C03633=1059.464,137.900,419.147,172.001,31.225,155.799
C03634=1059.459,137.652,419.168,172.000,31.222,155.799
C03635=1059.452,137.402,419.188,171.998,31.219,155.798
C03636=1059.447,137.154,419.210,171.997,31.217,155.798
C03637=1059.441,136.904,419.231,171.995,31.214,155.797
C03638=1059.435,136.656,419.251,171.993,31.211,155.797
C03639=1059.429,136.406,419.272,171.991,31.209,155.797
C03640=1059.423,136.157,419.293,171.989,31.206,155.796
C03641=1059.417,135.909,419.313,171.987,31.203,155.796
C03642=1059.411,135.659,419.334,171.986,31.201,155.795
C03643=1059.405,135.411,419.355,171.984,31.198,155.795
C03644=1059.399,135.161,419.376,171.983,31.196,155.794
C03645=1059.394,134.912,419.397,171.981,31.193,155.794
C03646=1059.387,134.663,419.417,171.979,31.190,155.794
C03647=1059.382,134.414,419.438,171.977,31.188,155.793
C03648=1059.376,134.165,419.459,171.976,31.185,155.793
C03649=1059.370,133.916,419.480,171.974,31.182,155.792
C03650=1059.364,133.666,419.500,171.972,31.180,155.792
C03651=1059.357,133.418,419.521,171.970,31.177,155.792
C03652=1059.352,133.168,419.542,171.968,31.174,155.791
C03653=1059.347,132.919,419.562,171.967,31.172,155.791
C03654=1059.340,132.670,419.583,171.966,31.169,155.790
C03655=1059.335,132.421,419.604,171.964,31.167,155.790
C03656=1059.330,132.172,419.624,171.962,31.164,155.789
C03657=1059.323,131.923,419.645,171.960,31.161,155.789
C03658=1059.317,131.674,419.666,171.958,31.159,155.789
C03659=1059.311,131.425,419.686,171.956,31.157,155.788
C03660=1059.305,131.176,419.706,171.955,31.154,155.788
C03661=1059.299,130.927,419.728,171.954,31.151,155.787
C03662=1059.293,130.678,419.748,171.952,31.149,155.787
C03663=1059.287,130.429,419.768,171.950,31.146,155.787
C03664=1059.281,130.179,419.789,171.948,31.143,155.786
C03665=1059.275,129.930,419.809,171.946,31.141,155.786
C03666=1059.270,129.681,419.829,171.945,31.139,155.785
C03667=1059.263,129.432,419.850,171.943,31.136,155.785
C03668=1059.257,129.184,419.870,171.941,31.133,155.785
C03669=1059.251,128.934,419.891,171.939,31.131,155.784
C03670=1059.245,128.685,419.911,171.938,31.128,155.784
C03671=1059.239,128.436,419.931,171.936,31.126,155.783
C03672=1059.233,128.186,419.952,171.935,31.123,155.783
C03673=1059.227,127.937,419.972,171.933,31.120,155.783
C03674=1059.221,127.689,419.993,171.931,31.118,155.782
C03675=1059.215,127.439,420.014,171.929,31.116,155.782
C03676=1059.209,127.191,420.034,171.927,31.113,155.781
C03677=1059.203,126.942,420.054,171.926,31.110,155.781
C03678=1059.197,126.716,420.072,171.925,31.108,155.781
C03679=1059.192,126.489,420.091,171.923,31.106,155.780
C03680=1059.187,126.265,420.109,171.921,31.103,155.780
C03681=1059.181,126.039,420.128,171.920,31.101,155.780
C03682=1059.175,125.813,420.146,171.918,31.098,155.779
C03683=1059.170,125.587,420.164,171.916,31.096,155.779
C03684=1059.164,125.361,420.182,171.915,31.094,155.778
C03685=1059.160,125.136,420.200,171.914,31.092,155.778
C03686=1059.153,124.887,420.221,171.912,31.089,155.778
C03687=1059.147,124.638,420.241,171.910,31.086,155.777
C03688=1059.142,124.389,420.262,171.909,31.084,155.777
C03689=1059.136,124.139,420.282,171.907,31.081,155.776
C03690=1059.130,123.890,420.302,171.905,31.079,155.776
C03691=1059.124,123.641,420.322,171.904,31.076,155.776
C03692=1059.118,123.392,420.342,171.902,31.073,155.775
C03693=1059.112,123.143,420.362,171.900,31.071,155.775
C03694=1059.106,122.894,420.382,171.898,31.069,155.774
C03695=1059.100,122.645,420.403,171.897,31.066,155.774
C03696=1059.094,122.396,420.423,171.895,31.063,155.774
C03697=1059.088,122.146,420.443,171.894,31.061,155.773
C03698=1059.082,121.897,420.463,171.892,31.058,155.773
C03699=1059.077,121.648,420.484,171.890,31.055,155.772
C03700=1059.071,121.399,420.504,171.888,31.053,155.772
C03701=1059.065,121.151,420.524,171.887,31.050,155.772
C03702=1059.058,120.901,420.544,171.886,31.048,155.771
C03703=1059.053,120.651,420.564,171.884,31.045,155.771
C03704=1059.047,120.403,420.584,171.882,31.042,155.770
C03705=1059.041,120.154,420.604,171.880,31.040,155.770
C03706=1059.033,119.822,420.631,171.878,31.036,155.769
C03707=1059.026,119.491,420.657,171.876,31.033,155.769
C03708=1059.018,119.158,420.684,171.874,31.030,155.768
C03709=1059.010,118.828,420.711,171.872,31.026,155.768
C03710=1059.004,118.578,420.731,171.870,31.024,155.767
C03711=1058.999,118.329,420.750,171.868,31.021,155.767
C03712=1058.992,118.080,420.771,171.867,31.018,155.767
C03713=1058.986,117.831,420.791,171.865,31.016,155.766
C03714=1058.981,117.582,420.811,171.864,31.013,155.766
C03715=1058.975,117.333,420.831,171.862,31.011,155.765
C03716=1058.969,117.083,420.850,171.860,31.008,155.765
C03717=1058.963,116.835,420.870,171.858,31.005,155.764
C03718=1058.957,116.586,420.890,171.857,31.003,155.764
C03719=1058.951,116.336,420.911,171.855,31.000,155.764
C03720=1058.946,116.086,420.931,171.854,30.997,155.763
C03721=1058.940,115.838,420.950,171.852,30.995,155.763
C03722=1058.934,115.589,420.970,171.850,30.992,155.762
C03723=1058.928,115.339,420.990,171.849,30.989,155.762
C03724=1058.923,115.090,421.010,171.847,30.987,155.762
C03725=1058.917,114.841,421.030,171.846,30.984,155.761
C03726=1058.911,114.592,421.049,171.844,30.981,155.761
C03727=1058.905,114.343,421.069,171.842,30.979,155.760
C03728=1058.900,114.094,421.090,171.840,30.976,155.760
C03729=1058.893,113.844,421.110,171.839,30.973,155.759
C03730=1058.887,113.595,421.130,171.838,30.971,155.759
C03731=1058.882,113.346,421.149,171.836,30.969,155.759
C03732=1058.875,113.097,421.168,171.834,30.966,155.758
C03733=1058.869,112.848,421.188,171.832,30.964,155.758
C03734=1058.863,112.599,421.207,171.830,30.961,155.758
C03735=1058.857,112.350,421.227,171.830,30.958,155.757
C03736=1058.852,112.101,421.247,171.828,30.956,155.757
C03737=1058.845,111.851,421.267,171.826,30.953,155.756
C03738=1058.839,111.602,421.286,171.824,30.950,155.756
C03739=1058.833,111.353,421.306,171.822,30.948,155.756
C03740=1058.828,111.104,421.325,171.822,30.946,155.755
C03741=1058.822,110.855,421.345,171.820,30.943,155.755
C03742=1058.815,110.570,421.367,171.818,30.940,155.754
C03743=1058.808,110.285,421.390,171.816,30.937,155.754
C03744=1058.801,110.000,421.412,171.814,30.934,155.753
C03745=1058.794,109.716,421.435,171.813,30.932,155.753
C03746=1058.788,109.467,421.454,171.811,30.929,155.753
C03747=1058.782,109.217,421.473,171.809,30.926,155.752
C03748=1058.776,108.968,421.493,171.807,30.924,155.752
C03749=1058.771,108.719,421.512,171.805,30.921,155.751
C03750=1058.764,108.469,421.533,171.804,30.919,155.751
C03751=1058.758,108.220,421.551,171.803,30.916,155.751
C03752=1058.752,107.971,421.571,171.801,30.914,155.750
C03753=1058.746,107.722,421.590,171.799,30.911,155.750
C03754=1058.740,107.473,421.610,171.797,30.908,155.749
C03755=1058.734,107.224,421.630,171.796,30.906,155.749
C03756=1058.729,106.974,421.649,171.795,30.904,155.749
C03757=1058.722,106.725,421.668,171.793,30.901,155.748
C03758=1058.716,106.476,421.688,171.791,30.898,155.748
C03759=1058.710,106.227,421.707,171.790,30.896,155.747
C03760=1058.705,105.978,421.726,171.788,30.893,155.747
C03761=1058.699,105.729,421.746,171.786,30.891,155.747
C03762=1058.692,105.480,421.765,171.785,30.888,155.746
C03763=1058.687,105.230,421.784,171.783,30.886,155.746
C03764=1058.681,104.981,421.804,171.782,30.883,155.745
C03765=1058.675,104.732,421.823,171.780,30.881,155.745
C03766=1058.669,104.483,421.842,171.778,30.878,155.745
C03767=1058.663,104.234,421.862,171.777,30.875,155.744
C03768=1058.657,103.985,421.881,171.776,30.873,155.744
C03769=1058.651,103.735,421.900,171.774,30.871,155.743
C03770=1058.645,103.486,421.919,171.772,30.868,155.743
C03771=1058.639,103.237,421.939,171.770,30.865,155.743
C03772=1058.633,102.988,421.958,171.769,30.863,155.742
C03773=1058.627,102.738,421.977,171.768,30.860,155.742
C03774=1058.622,102.489,421.996,171.766,30.857,155.741
C03775=1058.615,102.240,422.016,171.764,30.855,155.741
C03776=1058.609,101.991,422.035,171.762,30.853,155.741
C03777=1058.604,101.742,422.054,171.761,30.850,155.740
C03778=1058.598,101.492,422.074,171.760,30.847,155.740
C03779=1058.591,101.243,422.092,171.758,30.845,155.739
C03780=1058.585,100.994,422.112,171.756,30.842,155.739
C03781=1058.580,100.745,422.131,171.755,30.840,155.739
C03782=1058.573,100.496,422.150,171.753,30.837,155.738
C03783=1058.568,100.247,422.169,171.752,30.835,155.738
C03784=1058.563,99.997,422.188,171.750,30.832,155.737
C03785=1058.556,99.748,422.207,171.748,30.829,155.737
C03786=1058.550,99.499,422.226,171.747,30.827,155.737
C03787=1058.544,99.250,422.245,171.745,30.825,155.736
C03788=1058.538,99.001,422.265,171.743,30.822,155.736
C03789=1058.532,98.752,422.283,171.742,30.819,155.736
C03790=1058.526,98.502,422.303,171.741,30.817,155.735
C03791=1058.520,98.253,422.321,171.739,30.815,155.735
C03792=1058.514,98.004,422.340,171.737,30.812,155.734
C03793=1058.507,97.755,422.359,171.735,30.809,155.734
C03794=1058.502,97.505,422.378,171.735,30.807,155.734
C03795=1058.495,97.256,422.397,171.733,30.805,155.733
C03796=1058.490,97.007,422.416,171.731,30.802,155.733
C03797=1058.483,96.758,422.435,171.729,30.799,155.732
C03798=1058.477,96.508,422.454,171.728,30.797,155.732
C03799=1058.471,96.259,422.473,171.727,30.794,155.732
C03800=1058.466,96.010,422.492,171.725,30.792,155.731
C03801=1058.460,95.761,422.510,171.723,30.789,155.731
C03802=1058.454,95.512,422.530,171.721,30.787,155.730
C03803=1058.447,95.263,422.548,171.720,30.784,155.730
C03804=1058.442,95.013,422.567,171.719,30.781,155.730
C03805=1058.435,94.764,422.586,171.717,30.779,155.729
C03806=1058.428,94.479,422.608,171.715,30.776,155.729
C03807=1058.422,94.195,422.630,171.713,30.773,155.728
C03808=1058.415,93.910,422.650,171.711,30.771,155.728
C03809=1058.408,93.625,422.672,171.710,30.767,155.727
C03810=1058.403,93.376,422.691,171.708,30.765,155.727
C03811=1058.397,93.127,422.710,171.707,30.763,155.727
C03812=1058.391,92.877,422.729,171.705,30.760,155.726
C03813=1058.384,92.628,422.748,171.703,30.757,155.726
C03814=1058.379,92.379,422.767,171.702,30.755,155.726
C03815=1058.372,92.130,422.786,171.701,30.752,155.725
C03816=1058.367,91.881,422.803,171.699,30.750,155.725
C03817=1058.361,91.631,422.822,171.697,30.747,155.724
C03818=1058.355,91.382,422.841,171.696,30.745,155.724
C03819=1058.349,91.133,422.860,171.695,30.742,155.724
C03820=1058.343,90.883,422.879,171.693,30.740,155.723
C03821=1058.338,90.635,422.898,171.691,30.737,155.723
C03822=1058.331,90.385,422.916,171.690,30.735,155.722
C03823=1058.325,90.136,422.934,171.688,30.732,155.722
C03824=1058.319,89.886,422.954,171.686,30.730,155.722
C03825=1058.313,89.637,422.972,171.685,30.727,155.721
C03826=1058.307,89.388,422.990,171.684,30.725,155.721
C03827=1058.300,89.138,423.009,171.682,30.722,155.720
C03828=1058.295,88.890,423.027,171.680,30.720,155.720
C03829=1058.289,88.641,423.046,171.678,30.717,155.720
C03830=1058.283,88.391,423.064,171.678,30.715,155.719
C03831=1058.276,88.142,423.083,171.676,30.712,155.719
C03832=1058.270,87.893,423.102,171.674,30.710,155.719
C03833=1058.265,87.643,423.120,171.672,30.707,155.718
C03834=1058.259,87.394,423.139,171.671,30.705,155.718
C03835=1058.252,87.145,423.157,171.670,30.703,155.718
C03836=1058.246,86.896,423.176,171.668,30.700,155.717
C03837=1058.240,86.646,423.194,171.666,30.697,155.717
C03838=1058.235,86.397,423.213,171.665,30.695,155.716
C03839=1058.228,86.148,423.231,171.663,30.693,155.716
C03840=1058.222,85.899,423.249,171.662,30.690,155.716
C03841=1058.216,85.649,423.268,171.660,30.687,155.715
C03842=1058.210,85.400,423.286,171.659,30.685,155.715
C03843=1058.204,85.151,423.305,171.657,30.683,155.714
C03844=1058.198,84.902,423.323,171.655,30.680,155.714
C03845=1058.192,84.652,423.341,171.654,30.677,155.714
C03846=1058.185,84.403,423.360,171.653,30.675,155.713
C03847=1058.180,84.154,423.377,171.651,30.673,155.713
C03848=1058.174,83.904,423.397,171.649,30.670,155.713
C03849=1058.168,83.655,423.415,171.647,30.667,155.712
C03850=1058.162,83.406,423.433,171.647,30.665,155.712
C03851=1058.156,83.157,423.452,171.645,30.663,155.711
C03852=1058.150,82.907,423.469,171.643,30.660,155.711
C03853=1058.143,82.658,423.488,171.641,30.657,155.711
C03854=1058.139,82.409,423.506,171.640,30.655,155.710
C03855=1058.132,82.160,423.525,171.639,30.653,155.710
C03856=1058.126,81.910,423.543,171.637,30.650,155.709
C03857=1058.120,81.662,423.561,171.636,30.647,155.709
C03858=1058.114,81.412,423.579,171.634,30.645,155.709
C03859=1058.108,81.163,423.598,171.632,30.643,155.708
C03860=1058.102,80.913,423.616,171.631,30.640,155.708
C03861=1058.096,80.664,423.635,171.630,30.637,155.707
C03862=1058.090,80.415,423.652,171.628,30.635,155.707
C03863=1058.084,80.165,423.671,171.626,30.632,155.707
C03864=1058.078,79.916,423.689,171.624,30.630,155.706
C03865=1058.072,79.667,423.707,171.624,30.627,155.706
C03866=1058.066,79.418,423.725,171.622,30.625,155.706
C03867=1058.061,79.169,423.744,171.620,30.622,155.705
C03868=1058.055,78.919,423.762,171.619,30.620,155.705
C03869=1058.049,78.671,423.780,171.617,30.617,155.704
C03870=1058.041,78.385,423.801,171.616,30.614,155.704
C03871=1058.035,78.101,423.821,171.614,30.611,155.703
C03872=1058.028,77.815,423.842,171.612,30.608,155.703
C03873=1058.021,77.531,423.862,171.610,30.606,155.703
C03874=1058.014,77.282,423.881,171.609,30.603,155.702
C03875=1058.008,77.032,423.899,171.607,30.601,155.702
C03876=1058.003,76.783,423.916,171.606,30.598,155.702
C03877=1057.996,76.534,423.935,171.604,30.596,155.701
C03878=1057.990,76.284,423.953,171.602,30.594,155.701
C03879=1057.985,76.035,423.971,171.601,30.591,155.700
C03880=1057.978,75.786,423.989,171.600,30.588,155.700
C03881=1057.973,75.537,424.007,171.598,30.586,155.700
C03882=1057.967,75.287,424.025,171.596,30.584,155.699
C03883=1057.961,75.037,424.043,171.595,30.581,155.699
C03884=1057.955,74.789,424.061,171.594,30.578,155.698
C03885=1057.948,74.540,424.078,171.592,30.576,155.698
C03886=1057.942,74.290,424.096,171.590,30.573,155.698
C03887=1057.936,74.041,424.115,171.589,30.571,155.697
C03888=1057.930,73.792,424.132,171.587,30.569,155.697
C03889=1057.924,73.543,424.150,171.586,30.566,155.697
C03890=1057.918,73.293,424.168,171.584,30.563,155.696
C03891=1057.912,73.043,424.186,171.583,30.561,155.696
C03892=1057.906,72.795,424.204,171.581,30.559,155.696
C03893=1057.900,72.545,424.222,171.579,30.556,155.695
C03894=1057.894,72.296,424.239,171.579,30.553,155.695
C03895=1057.888,72.047,424.257,171.577,30.551,155.694
C03896=1057.882,71.797,424.275,171.575,30.549,155.694
C03897=1057.876,71.548,424.293,171.573,30.546,155.694
C03898=1057.870,71.299,424.311,171.572,30.544,155.693
C03899=1057.864,71.050,424.329,171.571,30.541,155.693
C03900=1057.858,70.800,424.347,171.569,30.539,155.693
C03901=1057.852,70.551,424.364,171.567,30.536,155.692
C03902=1057.846,70.301,424.382,171.566,30.534,155.692
C03903=1057.840,70.052,424.399,171.564,30.531,155.691
C03904=1057.834,69.803,424.418,171.563,30.529,155.691
C03905=1057.828,69.553,424.436,171.562,30.527,155.691
C03906=1057.821,69.305,424.453,171.560,30.524,155.690
C03907=1057.815,69.055,424.471,171.558,30.522,155.690
C03908=1057.810,68.806,424.488,171.556,30.519,155.690
C03909=1057.804,68.556,424.506,171.556,30.516,155.689
C03910=1057.797,68.308,424.523,171.554,30.514,155.689
C03911=1057.791,68.058,424.541,171.552,30.512,155.688
C03912=1057.786,67.809,424.559,171.551,30.509,155.688
C03913=1057.780,67.559,424.577,171.549,30.507,155.688
C03914=1057.773,67.310,424.594,171.548,30.504,155.687
C03915=1057.767,67.061,424.611,171.546,30.502,155.687
C03916=1057.761,66.811,424.629,171.545,30.500,155.687
C03917=1057.755,66.562,424.646,171.543,30.497,155.686
C03918=1057.749,66.312,424.664,171.542,30.494,155.686
C03919=1057.743,66.063,424.682,171.540,30.492,155.686
C03920=1057.736,65.814,424.699,171.539,30.490,155.685
C03921=1057.731,65.565,424.717,171.537,30.487,155.685
C03922=1057.725,65.315,424.735,171.535,30.485,155.684
C03923=1057.718,65.066,424.752,171.535,30.482,155.684
C03924=1057.712,64.817,424.770,171.533,30.480,155.684
C03925=1057.707,64.568,424.787,171.531,30.477,155.683
C03926=1057.700,64.318,424.804,171.529,30.475,155.683
C03927=1057.694,64.069,424.822,171.528,30.473,155.683
C03928=1057.688,63.820,424.839,171.527,30.470,155.682
C03929=1057.682,63.571,424.857,171.525,30.468,155.682
C03930=1057.675,63.321,424.874,171.523,30.465,155.681
C03931=1057.670,63.072,424.891,171.522,30.463,155.681
C03932=1057.663,62.822,424.908,171.520,30.460,155.681
C03933=1057.657,62.573,424.925,171.519,30.458,155.680
C03934=1057.650,62.288,424.946,171.517,30.456,155.680
C03935=1057.642,62.003,424.965,171.515,30.453,155.680
C03936=1057.636,61.719,424.985,171.513,30.450,155.679
C03937=1057.628,61.433,425.005,171.512,30.447,155.679
C03938=1057.623,61.184,425.022,171.511,30.445,155.678
C03939=1057.616,60.934,425.040,171.509,30.442,155.678
C03940=1057.610,60.685,425.057,171.507,30.440,155.678
C03941=1057.604,60.435,425.074,171.505,30.437,155.677
C03942=1057.597,60.187,425.091,171.505,30.435,155.677
C03943=1057.591,59.937,425.109,171.503,30.433,155.677
C03944=1057.585,59.688,425.126,171.501,30.431,155.676
C03945=1057.580,59.439,425.143,171.499,30.428,155.676
C03946=1057.573,59.189,425.160,171.498,30.426,155.676
C03947=1057.567,58.940,425.177,171.497,30.423,155.675
C03948=1057.561,58.691,425.195,171.495,30.421,155.675
C03949=1057.555,58.441,425.211,171.493,30.418,155.675
C03950=1057.548,58.192,425.229,171.492,30.416,155.674
C03951=1057.542,57.943,425.246,171.490,30.414,155.674
C03952=1057.536,57.693,425.263,171.489,30.411,155.673
C03953=1057.530,57.444,425.280,171.488,30.409,155.673
C03954=1057.524,57.195,425.297,171.486,30.406,155.673
C03955=1057.518,56.945,425.314,171.484,30.404,155.672
C03956=1057.512,56.696,425.331,171.483,30.401,155.672
C03957=1057.505,56.446,425.349,171.482,30.399,155.672
C03958=1057.500,56.197,425.366,171.480,30.397,155.671
C03959=1057.493,55.948,425.383,171.478,30.394,155.671
C03960=1057.487,55.699,425.400,171.476,30.392,155.671
C03961=1057.481,55.449,425.417,171.476,30.389,155.670
C03962=1057.475,55.200,425.434,171.474,30.387,155.670
C03963=1057.468,54.951,425.451,171.472,30.384,155.670
C03964=1057.463,54.701,425.468,171.470,30.382,155.669
C03965=1057.456,54.452,425.485,171.469,30.380,155.669
C03966=1057.451,54.202,425.502,171.468,30.377,155.668
C03967=1057.445,53.953,425.519,171.466,30.375,155.668
C03968=1057.438,53.704,425.536,171.465,30.372,155.668
C03969=1057.433,53.454,425.553,171.463,30.370,155.667
C03970=1057.426,53.205,425.571,171.462,30.367,155.667
C03971=1057.420,52.955,425.587,171.460,30.365,155.667
C03972=1057.414,52.706,425.604,171.459,30.363,155.666
C03973=1057.408,52.456,425.621,171.457,30.360,155.666
C03974=1057.402,52.208,425.638,171.455,30.358,155.666
C03975=1057.396,51.958,425.655,171.454,30.355,155.665
C03976=1057.390,51.709,425.672,171.453,30.353,155.665
C03977=1057.384,51.459,425.688,171.451,30.351,155.664
C03978=1057.378,51.210,425.706,171.449,30.348,155.664
C03979=1057.372,50.961,425.722,171.448,30.346,155.664
C03980=1057.365,50.711,425.740,171.447,30.343,155.663
C03981=1057.360,50.462,425.756,171.445,30.341,155.663
C03982=1057.354,50.213,425.773,171.443,30.338,155.663
C03983=1057.347,49.963,425.790,171.442,30.336,155.662
C03984=1057.342,49.714,425.808,171.441,30.334,155.662
C03985=1057.336,49.465,425.824,171.439,30.331,155.662
C03986=1057.329,49.216,425.841,171.437,30.329,155.661
C03987=1057.323,48.966,425.857,171.436,30.326,155.661
C03988=1057.317,48.717,425.875,171.434,30.324,155.661
C03989=1057.311,48.467,425.891,171.433,30.321,155.660
C03990=1057.305,48.218,425.908,171.432,30.319,155.660
C03991=1057.299,47.968,425.925,171.430,30.317,155.659
C03992=1057.293,47.719,425.942,171.428,30.314,155.659
C03993=1057.287,47.470,425.959,171.427,30.312,155.659
C03994=1057.282,47.221,425.976,171.426,30.309,155.658
C03995=1057.275,46.971,425.992,171.424,30.306,155.658
C03996=1057.269,46.722,426.009,171.422,30.304,155.658
C03997=1057.263,46.472,426.025,171.421,30.302,155.657
C03998=1057.257,46.187,426.045,171.420,30.299,155.657
C03999=1057.250,45.902,426.064,171.418,30.296,155.656
C04000=1057.243,45.617,426.084,171.416,30.294,155.656
C04001=1057.236,45.331,426.102,171.414,30.291,155.656
C04002=1057.230,45.082,426.119,171.413,30.288,155.655
C04003=1057.224,44.832,426.136,171.411,30.285,155.655
C04004=1057.219,44.583,426.152,171.409,30.283,155.655
C04005=1057.212,44.334,426.169,171.408,30.281,155.654
C04006=1057.206,44.085,426.185,171.407,30.278,155.654
C04007=1057.201,43.835,426.203,171.405,30.276,155.653
C04008=1057.195,43.585,426.219,171.404,30.273,155.653
C04009=1057.188,43.337,426.236,171.402,30.271,155.653
C04010=1057.182,43.087,426.252,171.401,30.268,155.652
C04011=1057.176,42.838,426.268,171.399,30.266,155.652
C04012=1057.170,42.588,426.285,171.398,30.264,155.652
C04013=1057.164,42.339,426.301,171.396,30.262,155.651
C04014=1057.158,42.090,426.318,171.394,30.259,155.651
C04015=1057.152,41.840,426.335,171.393,30.257,155.651
C04016=1057.146,41.591,426.351,171.392,30.254,155.650
C04017=1057.139,41.341,426.367,171.390,30.252,155.650
C04018=1057.133,41.092,426.384,171.388,30.249,155.650
C04019=1057.127,40.843,426.401,171.386,30.247,155.649
C04020=1057.121,40.594,426.417,171.386,30.245,155.649
C04021=1057.115,40.344,426.433,171.384,30.242,155.649
C04022=1057.109,40.095,426.449,171.382,30.240,155.648
C04023=1057.103,39.845,426.466,171.380,30.238,155.648
C04024=1057.097,39.596,426.482,171.380,30.235,155.647
C04025=1057.091,39.346,426.499,171.378,30.233,155.647
C04026=1057.085,39.097,426.515,171.376,30.230,155.647
C04027=1057.079,38.848,426.532,171.375,30.228,155.646
C04028=1057.073,38.598,426.549,171.373,30.225,155.646
C04029=1057.067,38.349,426.565,171.372,30.223,155.646
C04030=1057.061,38.099,426.582,171.370,30.220,155.645
C04031=1057.055,37.850,426.598,171.369,30.219,155.645
C04032=1057.048,37.601,426.613,171.367,30.216,155.645
C04033=1057.042,37.351,426.630,171.366,30.214,155.644
C04034=1057.036,37.102,426.646,171.364,30.212,155.644
C04035=1057.030,36.853,426.662,171.363,30.209,155.644
C04036=1057.024,36.603,426.679,171.361,30.207,155.643
C04037=1057.018,36.353,426.695,171.359,30.204,155.643
C04038=1057.011,36.104,426.711,171.358,30.202,155.643
C04039=1057.005,35.855,426.727,171.357,30.200,155.642
C04040=1056.999,35.605,426.743,171.355,30.197,155.642
C04041=1056.993,35.356,426.760,171.353,30.195,155.642
C04042=1056.987,35.107,426.776,171.352,30.192,155.641
C04043=1056.981,34.857,426.792,171.351,30.190,155.641
C04044=1056.974,34.608,426.808,171.349,30.188,155.641
C04045=1056.968,34.358,426.824,171.347,30.185,155.640
C04046=1056.962,34.109,426.841,171.345,30.183,155.640
C04047=1056.956,33.860,426.857,171.345,30.181,155.640
C04048=1056.950,33.610,426.873,171.343,30.179,155.639
C04049=1056.944,33.361,426.889,171.341,30.176,155.639
C04050=1056.938,33.111,426.904,171.339,30.174,155.639
C04051=1056.932,32.862,426.921,171.339,30.172,155.638
C04052=1056.926,32.613,426.937,171.337,30.169,155.638
C04053=1056.920,32.363,426.953,171.335,30.167,155.638
C04054=1056.913,32.114,426.969,171.333,30.164,155.637
C04055=1056.907,31.864,426.985,171.332,30.162,155.637
C04056=1056.901,31.615,427.002,171.331,30.160,155.637
C04057=1056.895,31.365,427.018,171.329,30.157,155.636
C04058=1056.889,31.116,427.033,171.327,30.155,155.636
C04059=1056.883,30.866,427.049,171.325,30.152,155.636
C04060=1056.877,30.617,427.065,171.325,30.150,155.635
C04061=1056.871,30.368,427.082,171.323,30.148,155.635
C04062=1056.864,30.082,427.100,171.321,30.146,155.635
C04063=1056.856,29.797,427.118,171.319,30.143,155.634
C04064=1056.849,29.512,427.137,171.318,30.140,155.634
C04065=1056.843,29.227,427.154,171.316,30.137,155.633
C04066=1056.837,28.978,427.171,171.314,30.135,155.633
C04067=1056.831,28.728,427.186,171.312,30.132,155.633
C04068=1056.824,28.478,427.202,171.312,30.130,155.632
C04069=1056.818,28.229,427.219,171.310,30.128,155.632
C04070=1056.811,27.980,427.234,171.308,30.126,155.632
C04071=1056.806,27.730,427.250,171.306,30.123,155.632
C04072=1056.800,27.481,427.266,171.305,30.121,155.631
C04073=1056.793,27.232,427.282,171.304,30.119,155.631
C04074=1056.788,26.982,427.297,171.302,30.117,155.631
C04075=1056.782,26.732,427.313,171.300,30.114,155.630
C04076=1056.775,26.483,427.329,171.299,30.112,155.630
C04077=1056.769,26.233,427.345,171.298,30.110,155.630
C04078=1056.763,25.984,427.360,171.296,30.107,155.629
C04079=1056.757,25.735,427.377,171.294,30.105,155.629
C04080=1056.750,25.485,427.392,171.292,30.103,155.629
C04081=1056.744,25.236,427.408,171.291,30.100,155.628
C04082=1056.738,24.986,427.424,171.290,30.098,155.628
C04083=1056.732,24.737,427.439,171.288,30.096,155.628
C04084=1056.726,24.487,427.455,171.286,30.094,155.627
C04085=1056.719,24.238,427.471,171.285,30.091,155.627
C04086=1056.714,23.988,427.486,171.284,30.089,155.627
C04087=1056.707,23.739,427.502,171.282,30.087,155.626
C04088=1056.701,23.489,427.518,171.280,30.084,155.626
C04089=1056.695,23.240,427.533,171.279,30.082,155.626
C04090=1056.690,22.991,427.548,171.277,30.080,155.625
C04091=1056.683,22.742,427.564,171.276,30.077,155.625
C04092=1056.677,22.493,427.580,171.274,30.075,155.625
C04093=1056.671,22.243,427.595,171.272,30.073,155.624
C04094=1056.665,21.994,427.612,171.271,30.070,155.624
C04095=1056.659,21.744,427.627,171.270,30.068,155.624
C04096=1056.652,21.495,427.643,171.268,30.066,155.623
C04097=1056.647,21.245,427.658,171.266,30.063,155.623
C04098=1056.640,20.996,427.674,171.265,30.061,155.623
C04099=1056.634,20.746,427.690,171.264,30.059,155.622
C04100=1056.628,20.497,427.705,171.262,30.057,155.622
C04101=1056.622,20.247,427.721,171.260,30.054,155.622
C04102=1056.615,19.998,427.736,171.258,30.052,155.622
C04103=1056.610,19.748,427.752,171.257,30.050,155.621
C04104=1056.604,19.499,427.767,171.256,30.047,155.621
C04105=1056.597,19.250,427.782,171.254,30.045,155.621
C04106=1056.591,19.000,427.798,171.252,30.043,155.620
C04107=1056.585,18.751,427.813,171.251,30.041,155.620
C04108=1056.579,18.501,427.829,171.250,30.038,155.620
C04109=1056.573,18.252,427.845,171.248,30.036,155.619
C04110=1056.566,18.002,427.860,171.246,30.034,155.619
C04111=1056.560,17.753,427.876,171.244,30.032,155.619
C04112=1056.554,17.503,427.891,171.244,30.029,155.618
C04113=1056.548,17.254,427.905,171.242,30.027,155.618
C04114=1056.542,17.005,427.922,171.240,30.025,155.618
C04115=1056.536,16.755,427.937,171.238,30.023,155.617
C04116=1056.530,16.506,427.953,171.237,30.020,155.617
C04117=1056.523,16.256,427.968,171.236,30.018,155.617
C04118=1056.517,16.006,427.983,171.234,30.016,155.616
C04119=1056.511,15.757,427.999,171.232,30.014,155.616
C04120=1056.505,15.508,428.013,171.230,30.011,155.616
C04121=1056.499,15.258,428.028,171.230,30.009,155.615
C04122=1056.493,15.009,428.045,171.228,30.007,155.615
C04123=1056.487,14.759,428.060,171.226,30.005,155.615
C04124=1056.481,14.510,428.075,171.224,30.002,155.615
C04125=1056.474,14.260,428.090,171.223,30.000,155.614
C04126=1056.468,13.977,428.108,171.221,29.997,155.614
C04127=1056.460,13.692,428.125,171.219,29.995,155.614
C04128=1056.453,13.409,428.143,171.217,29.993,155.613
C04129=1056.446,13.124,428.160,171.216,29.990,155.613
C04130=1056.440,12.875,428.174,171.214,29.988,155.613
C04131=1056.434,12.626,428.189,171.213,29.986,155.612
C04132=1056.427,12.376,428.205,171.211,29.983,155.612
C04133=1056.421,12.127,428.220,171.209,29.981,155.612
C04134=1056.414,11.877,428.235,171.208,29.979,155.611
C04135=1056.408,11.627,428.250,171.206,29.976,155.611
C04136=1056.402,11.378,428.265,171.205,29.974,155.611
C04137=1056.396,11.129,428.281,171.203,29.972,155.611
C04138=1056.390,10.880,428.296,171.202,29.970,155.610
C04139=1056.383,10.630,428.311,171.200,29.968,155.610
C04140=1056.377,10.380,428.326,171.198,29.966,155.610
C04141=1056.371,10.131,428.341,171.196,29.964,155.609
C04142=1056.365,9.882,428.355,171.195,29.962,155.609
C04143=1056.358,9.633,428.371,171.194,29.959,155.609
C04144=1056.353,9.383,428.386,171.192,29.957,155.608
C04145=1056.346,9.133,428.401,171.190,29.955,155.608
C04146=1056.340,8.883,428.416,171.188,29.952,155.608
C04147=1056.334,8.634,428.431,171.188,29.950,155.608
C04148=1056.328,8.385,428.446,171.186,29.948,155.607
C04149=1056.321,8.135,428.461,171.184,29.946,155.607
C04150=1056.315,7.885,428.476,171.182,29.944,155.607
C04151=1056.309,7.636,428.490,171.180,29.942,155.606
C04152=1056.303,7.387,428.505,171.180,29.940,155.606
C04153=1056.296,7.137,428.520,171.178,29.938,155.606
C04154=1056.291,6.887,428.536,171.176,29.935,155.605
C04155=1056.285,6.639,428.551,171.174,29.933,155.605
C04156=1056.278,6.389,428.566,171.173,29.931,155.605
C04157=1056.272,6.139,428.581,171.171,29.928,155.605
C04158=1056.265,5.890,428.596,171.170,29.926,155.604
C04159=1056.260,5.641,428.610,171.168,29.924,155.604
C04160=1056.253,5.391,428.625,171.167,29.922,155.604
C04161=1056.247,5.142,428.640,171.165,29.920,155.604
C04162=1056.241,4.892,428.655,171.163,29.918,155.603
C04163=1056.235,4.643,428.670,171.162,29.916,155.603
C04164=1056.228,4.393,428.685,171.160,29.913,155.603
C04165=1056.222,4.143,428.699,171.159,29.911,155.602
C04166=1056.217,3.894,428.714,171.157,29.909,155.602
C04167=1056.211,3.644,428.729,171.155,29.906,155.602
C04168=1056.204,3.394,428.744,171.153,29.904,155.601
C04169=1056.199,3.145,428.759,171.153,29.902,155.601
C04170=1056.192,2.896,428.774,171.151,29.900,155.601
C04171=1056.186,2.646,428.788,171.149,29.898,155.601
C04172=1056.180,2.397,428.803,171.147,29.896,155.600
C04173=1056.174,2.148,428.818,171.146,29.894,155.600
C04174=1056.167,1.898,428.833,171.144,29.891,155.600
C04175=1056.162,1.649,428.848,171.143,29.889,155.599
C04176=1056.155,1.399,428.862,171.141,29.887,155.599
C04177=1056.149,1.149,428.877,171.139,29.885,155.599
C04178=1056.143,0.900,428.891,171.138,29.882,155.598
C04179=1056.137,0.650,428.906,171.136,29.880,155.598
C04180=1056.131,0.401,428.921,171.135,29.878,155.598
C04181=1056.125,0.152,428.936,171.133,29.876,155.598
C04182=1056.118,-0.098,428.951,171.132,29.874,155.597
C04183=1056.113,-0.347,428.965,171.130,29.872,155.597
C04184=1056.107,-0.597,428.979,171.128,29.870,155.597
C04185=1056.101,-0.846,428.994,171.126,29.867,155.597
C04186=1056.094,-1.096,429.009,171.126,29.865,155.596
C04187=1056.088,-1.345,429.024,171.124,29.863,155.596
C04188=1056.082,-1.594,429.039,171.122,29.860,155.596
C04189=1056.076,-1.845,429.053,171.120,29.858,155.595
C04190=1056.069,-2.127,429.069,171.118,29.856,155.595
C04191=1056.063,-2.409,429.086,171.117,29.853,155.595
C04192=1056.056,-2.690,429.103,171.115,29.851,155.594
C04193=1056.050,-2.972,429.119,171.113,29.848,155.594
C04194=1056.043,-3.222,429.134,171.112,29.846,155.594
C04195=1056.037,-3.472,429.149,171.110,29.844,155.593
C04196=1056.031,-3.721,429.162,171.108,29.842,155.593
C04197=1056.024,-3.971,429.177,171.106,29.840,155.593
C04198=1056.018,-4.220,429.192,171.104,29.838,155.593
C04199=1056.012,-4.470,429.206,171.104,29.836,155.592
C04200=1056.005,-4.719,429.220,171.102,29.834,155.592
C04201=1055.999,-4.968,429.235,171.100,29.832,155.592
C04202=1055.993,-5.219,429.249,171.098,29.830,155.592
C04203=1055.987,-5.467,429.263,171.097,29.827,155.591
C04204=1055.981,-5.717,429.278,171.095,29.825,155.591
C04205=1055.974,-5.967,429.292,171.093,29.823,155.591
C04206=1055.969,-6.216,429.307,171.092,29.821,155.590
C04207=1055.962,-6.466,429.321,171.090,29.819,155.590
C04208=1055.956,-6.715,429.335,171.089,29.817,155.590
C04209=1055.950,-6.965,429.350,171.087,29.815,155.590
C04210=1055.943,-7.214,429.363,171.085,29.813,155.589
C04211=1055.937,-7.464,429.378,171.083,29.811,155.589
C04212=1055.931,-7.714,429.393,171.082,29.809,155.589
C04213=1055.925,-7.963,429.407,171.081,29.807,155.589
C04214=1055.918,-8.213,429.421,171.079,29.804,155.588
C04215=1055.913,-8.462,429.435,171.077,29.802,155.588
C04216=1055.907,-8.712,429.450,171.075,29.801,155.588
C04217=1055.900,-8.961,429.464,171.074,29.799,155.588
C04218=1055.894,-9.211,429.478,171.072,29.796,155.587
C04219=1055.888,-9.460,429.492,171.070,29.794,155.587
C04220=1055.881,-9.709,429.507,171.068,29.792,155.587
C04221=1055.876,-9.959,429.521,171.068,29.790,155.586
C04222=1055.869,-10.208,429.536,171.066,29.788,155.586
C04223=1055.864,-10.458,429.549,171.064,29.786,155.586
C04224=1055.857,-10.708,429.563,171.062,29.784,155.586
C04225=1055.851,-10.957,429.578,171.061,29.782,155.585
C04226=1055.845,-11.207,429.592,171.059,29.780,155.585
C04227=1055.839,-11.456,429.606,171.057,29.778,155.585
C04228=1055.832,-11.706,429.620,171.055,29.775,155.585
C04229=1055.827,-11.955,429.635,171.054,29.773,155.584
C04230=1055.820,-12.205,429.648,171.053,29.771,155.584
C04231=1055.814,-12.454,429.663,171.051,29.769,155.584
C04232=1055.809,-12.704,429.677,171.049,29.767,155.584
C04233=1055.802,-12.954,429.690,171.047,29.765,155.583
C04234=1055.796,-13.202,429.705,171.046,29.763,155.583
C04235=1055.789,-13.452,429.719,171.044,29.761,155.583
C04236=1055.783,-13.701,429.733,171.042,29.759,155.583
C04237=1055.777,-13.952,429.747,171.041,29.757,155.582
C04238=1055.771,-14.201,429.761,171.040,29.755,155.582
C04239=1055.765,-14.450,429.775,171.038,29.753,155.582
C04240=1055.759,-14.700,429.790,171.036,29.751,155.582
C04241=1055.753,-14.949,429.803,171.034,29.749,155.581
C04242=1055.747,-15.199,429.818,171.032,29.746,155.581
C04243=1055.740,-15.448,429.831,171.031,29.744,155.581
C04244=1055.734,-15.699,429.845,171.029,29.743,155.581
C04245=1055.728,-15.947,429.859,171.027,29.740,155.580
C04246=1055.722,-16.198,429.873,171.026,29.738,155.580
C04247=1055.716,-16.447,429.887,171.025,29.737,155.580
C04248=1055.710,-16.696,429.901,171.023,29.735,155.580
C04249=1055.703,-16.946,429.915,171.021,29.733,155.579
C04250=1055.697,-17.195,429.928,171.019,29.731,155.579
C04251=1055.691,-17.445,429.942,171.017,29.729,155.579
C04252=1055.684,-17.695,429.956,171.016,29.727,155.579
C04253=1055.678,-17.944,429.971,171.014,29.724,155.578
C04254=1055.671,-18.224,429.985,171.012,29.722,155.578
C04255=1055.664,-18.505,430.001,171.010,29.720,155.578
C04256=1055.657,-18.785,430.017,171.009,29.718,155.577
C04257=1055.650,-19.065,430.032,171.007,29.716,155.577
C04258=1055.644,-19.315,430.046,171.005,29.714,155.577
C04259=1055.638,-19.565,430.060,171.003,29.712,155.577
C04260=1055.631,-19.815,430.073,171.002,29.710,155.577
C04261=1055.625,-20.064,430.088,171.000,29.708,155.576
C04262=1055.619,-20.313,430.101,170.998,29.706,155.576
C04263=1055.612,-20.563,430.115,170.996,29.704,155.576
C04264=1055.607,-20.813,430.129,170.994,29.702,155.576
C04265=1055.601,-21.062,430.142,170.993,29.700,155.575
C04266=1055.595,-21.312,430.156,170.991,29.698,155.575
C04267=1055.588,-21.561,430.169,170.990,29.696,155.575
C04268=1055.582,-21.811,430.183,170.988,29.694,155.575
C04269=1055.576,-22.060,430.198,170.987,29.692,155.574
C04270=1055.570,-22.310,430.211,170.985,29.690,155.574
C04271=1055.564,-22.559,430.225,170.983,29.688,155.574
C04272=1055.557,-22.809,430.238,170.981,29.686,155.574
C04273=1055.551,-23.058,430.252,170.979,29.685,155.574
C04274=1055.546,-23.308,430.265,170.978,29.682,155.573
C04275=1055.539,-23.558,430.279,170.976,29.680,155.573
C04276=1055.533,-23.807,430.292,170.974,29.679,155.573
C04277=1055.527,-24.057,430.306,170.972,29.676,155.573
C04278=1055.521,-24.306,430.319,170.971,29.674,155.572
C04279=1055.514,-24.556,430.333,170.970,29.673,155.572
C04280=1055.509,-24.805,430.347,170.968,29.671,155.572
C04281=1055.502,-25.055,430.360,170.966,29.668,155.572
C04282=1055.496,-25.305,430.374,170.964,29.667,155.571
C04283=1055.490,-25.554,430.388,170.963,29.665,155.571
C04284=1055.484,-25.804,430.401,170.961,29.662,155.571
C04285=1055.478,-26.053,430.415,170.959,29.661,155.571
C04286=1055.472,-26.303,430.429,170.957,29.659,155.570
C04287=1055.465,-26.552,430.442,170.956,29.656,155.570
C04288=1055.460,-26.802,430.456,170.954,29.655,155.570
C04289=1055.454,-27.051,430.469,170.952,29.653,155.570
C04290=1055.447,-27.301,430.483,170.950,29.651,155.570
C04291=1055.441,-27.550,430.496,170.949,29.649,155.569
C04292=1055.434,-27.800,430.509,170.947,29.647,155.569
C04293=1055.428,-28.050,430.523,170.946,29.645,155.569
C04294=1055.422,-28.300,430.535,170.944,29.644,155.569
C04295=1055.416,-28.549,430.549,170.942,29.642,155.568
C04296=1055.410,-28.798,430.562,170.941,29.640,155.568
C04297=1055.403,-29.048,430.576,170.939,29.638,155.568
C04298=1055.397,-29.298,430.589,170.937,29.636,155.568
C04299=1055.391,-29.547,430.603,170.935,29.634,155.568
C04300=1055.385,-29.796,430.616,170.933,29.632,155.567
C04301=1055.378,-30.047,430.629,170.932,29.631,155.567
C04302=1055.372,-30.296,430.642,170.930,29.629,155.567
C04303=1055.366,-30.546,430.656,170.928,29.627,155.567
C04304=1055.360,-30.795,430.669,170.926,29.625,155.567
C04305=1055.354,-31.044,430.682,170.925,29.623,155.566
C04306=1055.347,-31.295,430.695,170.923,29.621,155.566
C04307=1055.341,-31.544,430.709,170.921,29.619,155.566
C04308=1055.335,-31.793,430.722,170.919,29.617,155.566
C04309=1055.329,-32.042,430.735,170.917,29.616,155.566
C04310=1055.322,-32.292,430.749,170.916,29.613,155.565
C04311=1055.316,-32.542,430.761,170.914,29.612,155.565
C04312=1055.310,-32.792,430.775,170.913,29.610,155.565
C04313=1055.304,-33.041,430.788,170.911,29.608,155.565
C04314=1055.298,-33.290,430.802,170.910,29.607,155.564
C04315=1055.292,-33.540,430.814,170.908,29.605,155.564
C04316=1055.285,-33.790,430.828,170.906,29.603,155.564
C04317=1055.279,-34.040,430.841,170.904,29.601,155.564
C04318=1055.273,-34.319,430.856,170.902,29.599,155.564
C04319=1055.266,-34.599,430.870,170.900,29.597,155.563
C04320=1055.259,-34.878,430.885,170.898,29.595,155.563
C04321=1055.252,-35.158,430.900,170.896,29.592,155.563
C04322=1055.246,-35.408,430.913,170.894,29.591,155.563
C04323=1055.240,-35.657,430.926,170.893,29.589,155.563
C04324=1055.234,-35.907,430.939,170.891,29.587,155.562
C04325=1055.227,-36.157,430.952,170.889,29.585,155.562
C04326=1055.221,-36.406,430.966,170.887,29.583,155.562
C04327=1055.215,-36.656,430.978,170.885,29.582,155.562
C04328=1055.209,-36.905,430.991,170.884,29.580,155.562
C04329=1055.203,-37.155,431.004,170.882,29.578,155.561
C04330=1055.197,-37.404,431.017,170.880,29.576,155.561
C04331=1055.190,-37.654,431.031,170.878,29.574,155.561
C04332=1055.184,-37.904,431.043,170.877,29.572,155.561
C04333=1055.178,-38.153,431.056,170.875,29.571,155.561
C04334=1055.172,-38.403,431.069,170.873,29.569,155.560
C04335=1055.166,-38.652,431.082,170.871,29.567,155.560
C04336=1055.160,-38.903,431.095,170.869,29.565,155.560
C04337=1055.153,-39.152,431.108,170.868,29.563,155.560
C04338=1055.147,-39.401,431.122,170.866,29.562,155.560
C04339=1055.141,-39.651,431.134,170.864,29.560,155.559
C04340=1055.134,-39.900,431.147,170.862,29.558,155.559
C04341=1055.128,-40.150,431.159,170.861,29.556,155.559
C04342=1055.122,-40.399,431.173,170.860,29.555,155.559
C04343=1055.116,-40.649,431.185,170.858,29.553,155.559
C04344=1055.110,-40.899,431.198,170.856,29.552,155.558
C04345=1055.103,-41.148,431.210,170.854,29.549,155.558
C04346=1055.097,-41.398,431.223,170.853,29.548,155.558
C04347=1055.091,-41.648,431.237,170.851,29.546,155.558
C04348=1055.085,-41.897,431.249,170.849,29.545,155.558
C04349=1055.079,-42.147,431.262,170.847,29.543,155.558
C04350=1055.072,-42.396,431.274,170.845,29.541,155.557
C04351=1055.066,-42.646,431.288,170.844,29.539,155.557
C04352=1055.060,-42.895,431.300,170.842,29.538,155.557
C04353=1055.054,-43.145,431.313,170.840,29.536,155.557
C04354=1055.048,-43.395,431.326,170.838,29.535,155.557
C04355=1055.041,-43.644,431.338,170.836,29.532,155.556
C04356=1055.035,-43.893,431.351,170.835,29.531,155.556
C04357=1055.029,-44.143,431.364,170.833,29.529,155.556
C04358=1055.023,-44.393,431.376,170.831,29.528,155.556
C04359=1055.017,-44.642,431.390,170.829,29.526,155.556
C04360=1055.010,-44.892,431.402,170.827,29.524,155.556
C04361=1055.004,-45.142,431.414,170.826,29.522,155.555
C04362=1054.998,-45.391,431.427,170.824,29.521,155.555
C04363=1054.992,-45.641,431.440,170.822,29.519,155.555
C04364=1054.985,-45.891,431.452,170.820,29.517,155.555
C04365=1054.979,-46.140,431.465,170.819,29.515,155.555
C04366=1054.973,-46.390,431.478,170.817,29.514,155.554
C04367=1054.967,-46.640,431.490,170.815,29.512,155.554
C04368=1054.962,-46.890,431.503,170.813,29.510,155.554
C04369=1054.955,-47.139,431.516,170.811,29.509,155.554
C04370=1054.949,-47.388,431.528,170.810,29.507,155.554
C04371=1054.943,-47.638,431.541,170.808,29.506,155.554
C04372=1054.937,-47.888,431.553,170.806,29.503,155.553
C04373=1054.930,-48.137,431.566,170.804,29.502,155.553
C04374=1054.925,-48.386,431.578,170.802,29.500,155.553
C04375=1054.919,-48.636,431.591,170.801,29.499,155.553
C04376=1054.913,-48.886,431.603,170.799,29.497,155.553
C04377=1054.906,-49.135,431.616,170.797,29.495,155.553
C04378=1054.900,-49.385,431.628,170.795,29.494,155.553
C04379=1054.894,-49.635,431.641,170.793,29.492,155.552
C04380=1054.887,-49.884,431.653,170.792,29.490,155.552
C04381=1054.881,-50.134,431.666,170.790,29.488,155.552
C04382=1054.875,-50.414,431.680,170.787,29.487,155.552
C04383=1054.868,-50.694,431.693,170.785,29.485,155.552
C04384=1054.861,-50.975,431.707,170.784,29.483,155.551
C04385=1054.854,-51.254,431.721,170.781,29.481,155.551
C04386=1054.847,-51.503,431.733,170.779,29.479,155.551
C04387=1054.841,-51.753,431.746,170.777,29.478,155.551
C04388=1054.834,-52.003,431.758,170.775,29.477,155.551
C04389=1054.828,-52.253,431.770,170.773,29.475,155.551
C04390=1054.822,-52.502,431.782,170.772,29.474,155.551
C04391=1054.816,-52.752,431.795,170.770,29.472,155.550
C04392=1054.809,-53.002,431.807,170.768,29.470,155.550
C04393=1054.803,-53.251,431.819,170.766,29.469,155.550
C04394=1054.797,-53.501,431.831,170.764,29.467,155.550
C04395=1054.790,-53.751,431.843,170.763,29.466,155.550
C04396=1054.784,-54.000,431.857,170.761,29.465,155.550
C04397=1054.777,-54.250,431.868,170.759,29.463,155.550
C04398=1054.771,-54.499,431.880,170.757,29.461,155.550
C04399=1054.765,-54.749,431.893,170.755,29.460,155.549
C04400=1054.759,-54.998,431.905,170.754,29.458,155.549
C04401=1054.753,-55.248,431.917,170.752,29.457,155.549
C04402=1054.746,-55.497,431.929,170.750,29.455,155.549
C04403=1054.739,-55.747,431.941,170.748,29.454,155.549
C04404=1054.734,-55.997,431.953,170.746,29.452,155.549
C04405=1054.727,-56.247,431.965,170.745,29.451,155.549
C04406=1054.721,-56.497,431.977,170.743,29.449,155.548
C04407=1054.715,-56.746,431.989,170.741,29.447,155.548
C04408=1054.709,-56.995,432.001,170.739,29.446,155.548
C04409=1054.703,-57.245,432.014,170.736,29.444,155.548
C04410=1054.696,-57.495,432.025,170.735,29.443,155.548
C04411=1054.689,-57.744,432.037,170.733,29.441,155.548
C04412=1054.683,-57.994,432.050,170.731,29.440,155.548
C04413=1054.677,-58.244,432.062,170.729,29.438,155.547
C04414=1054.671,-58.493,432.074,170.727,29.437,155.547
C04415=1054.665,-58.743,432.086,170.726,29.436,155.547
C04416=1054.658,-58.993,432.097,170.724,29.434,155.547
C04417=1054.653,-59.243,432.110,170.722,29.432,155.547
C04418=1054.646,-59.492,432.122,170.720,29.431,155.547
C04419=1054.640,-59.741,432.133,170.718,29.429,155.547
C04420=1054.634,-59.991,432.146,170.716,29.428,155.547
C04421=1054.627,-60.241,432.158,170.715,29.427,155.546
C04422=1054.621,-60.490,432.170,170.713,29.425,155.546
C04423=1054.615,-60.741,432.182,170.711,29.423,155.546
C04424=1054.609,-60.989,432.193,170.709,29.422,155.546
C04425=1054.602,-61.239,432.205,170.707,29.421,155.546
C04426=1054.596,-61.489,432.218,170.706,29.419,155.546
C04427=1054.590,-61.739,432.230,170.704,29.418,155.546
C04428=1054.584,-61.988,432.241,170.702,29.416,155.546
C04429=1054.578,-62.238,432.253,170.699,29.415,155.546
C04430=1054.572,-62.487,432.265,170.697,29.413,155.545
C04431=1054.565,-62.737,432.277,170.696,29.412,155.545
C04432=1054.560,-62.987,432.289,170.694,29.410,155.545
C04433=1054.553,-63.236,432.301,170.692,29.409,155.545
C04434=1054.547,-63.486,432.313,170.690,29.407,155.545
C04435=1054.541,-63.736,432.325,170.688,29.406,155.545
C04436=1054.535,-63.985,432.336,170.687,29.404,155.545
C04437=1054.528,-64.235,432.348,170.685,29.403,155.545
C04438=1054.522,-64.485,432.361,170.683,29.402,155.544
C04439=1054.517,-64.734,432.371,170.681,29.400,155.544
C04440=1054.510,-64.984,432.383,170.679,29.399,155.544
C04441=1054.503,-65.233,432.395,170.677,29.397,155.544
C04442=1054.498,-65.483,432.407,170.676,29.396,155.544
C04443=1054.492,-65.733,432.419,170.674,29.394,155.544
C04444=1054.485,-65.982,432.431,170.672,29.393,155.544
C04445=1054.480,-66.232,432.442,170.669,29.391,155.544
C04446=1054.472,-66.514,432.455,170.667,29.390,155.543
C04447=1054.466,-66.795,432.469,170.666,29.388,155.543
C04448=1054.459,-67.076,432.481,170.663,29.386,155.543
C04449=1054.452,-67.358,432.495,170.661,29.385,155.543
C04450=1054.446,-67.607,432.507,170.659,29.384,155.543
C04451=1054.440,-67.857,432.519,170.657,29.382,155.543
C04452=1054.434,-68.107,432.530,170.656,29.380,155.543
C04453=1054.427,-68.356,432.542,170.654,29.379,155.543
C04454=1054.422,-68.606,432.553,170.652,29.378,155.542
C04455=1054.416,-68.855,432.566,170.650,29.376,155.542
C04456=1054.409,-69.106,432.577,170.648,29.375,155.542
C04457=1054.403,-69.355,432.588,170.647,29.374,155.542
C04458=1054.397,-69.604,432.600,170.645,29.373,155.542
C04459=1054.392,-69.854,432.612,170.642,29.371,155.542
C04460=1054.385,-70.103,432.624,170.640,29.369,155.542
C04461=1054.379,-70.354,432.635,170.638,29.368,155.542
C04462=1054.373,-70.603,432.647,170.637,29.367,155.542
C04463=1054.367,-70.853,432.658,170.635,29.365,155.541
C04464=1054.361,-71.102,432.670,170.633,29.364,155.541
C04465=1054.355,-71.352,432.681,170.631,29.362,155.541
C04466=1054.348,-71.601,432.693,170.629,29.361,155.541
C04467=1054.343,-71.851,432.705,170.627,29.360,155.541
C04468=1054.337,-72.102,432.716,170.626,29.358,155.541
C04469=1054.331,-72.351,432.728,170.624,29.357,155.541
C04470=1054.324,-72.601,432.739,170.622,29.356,155.541
C04471=1054.318,-72.850,432.750,170.620,29.355,155.541
C04472=1054.313,-73.100,432.762,170.617,29.353,155.541
C04473=1054.306,-73.349,432.774,170.616,29.351,155.540
C04474=1054.300,-73.599,432.785,170.614,29.350,155.540
C04475=1054.294,-73.849,432.796,170.612,29.348,155.540
C04476=1054.288,-74.098,432.808,170.610,29.347,155.540
C04477=1054.282,-74.348,432.819,170.608,29.346,155.540
C04478=1054.275,-74.597,432.831,170.606,29.345,155.540
C04479=1054.269,-74.848,432.842,170.605,29.344,155.540
C04480=1054.263,-75.097,432.853,170.603,29.342,155.540
C04481=1054.257,-75.347,432.865,170.601,29.341,155.540
C04482=1054.251,-75.596,432.876,170.599,29.340,155.540
C04483=1054.245,-75.846,432.887,170.596,29.338,155.540
C04484=1054.239,-76.095,432.898,170.594,29.337,155.540
C04485=1054.232,-76.345,432.910,170.593,29.336,155.540
C04486=1054.226,-76.595,432.921,170.591,29.335,155.539
C04487=1054.220,-76.845,432.932,170.589,29.333,155.539
C04488=1054.214,-77.094,432.943,170.587,29.332,155.539
C04489=1054.208,-77.344,432.955,170.585,29.331,155.539
C04490=1054.202,-77.594,432.966,170.583,29.330,155.539
C04491=1054.195,-77.843,432.978,170.582,29.329,155.539
C04492=1054.190,-78.093,432.988,170.580,29.328,155.539
C04493=1054.183,-78.343,433.000,170.577,29.326,155.539
C04494=1054.177,-78.592,433.011,170.575,29.325,155.539
C04495=1054.171,-78.842,433.022,170.573,29.324,155.539
C04496=1054.165,-79.091,433.033,170.572,29.322,155.539
C04497=1054.159,-79.342,433.045,170.570,29.321,155.539
C04498=1054.153,-79.591,433.055,170.568,29.320,155.539
C04499=1054.147,-79.841,433.067,170.566,29.318,155.538
C04500=1054.140,-80.090,433.077,170.564,29.317,155.538
C04501=1054.134,-80.340,433.089,170.562,29.316,155.538
C04502=1054.128,-80.589,433.100,170.559,29.315,155.538
C04503=1054.121,-80.840,433.111,170.558,29.314,155.538
C04504=1054.115,-81.089,433.121,170.556,29.313,155.538
C04505=1054.109,-81.339,433.133,170.554,29.312,155.538
C04506=1054.103,-81.589,433.143,170.552,29.311,155.538
C04507=1054.096,-81.838,433.154,170.550,29.310,155.538
C04508=1054.090,-82.088,433.165,170.548,29.309,155.538
C04509=1054.083,-82.337,433.177,170.547,29.308,155.538
C04510=1054.077,-82.621,433.189,170.544,29.306,155.538
C04511=1054.069,-82.904,433.201,170.542,29.305,155.538
C04512=1054.062,-83.188,433.214,170.539,29.304,155.538
C04513=1054.056,-83.472,433.226,170.537,29.303,155.538
C04514=1054.049,-83.722,433.237,170.535,29.302,155.538
C04515=1054.043,-83.971,433.248,170.534,29.300,155.538
C04516=1054.037,-84.221,433.259,170.532,29.299,155.538
C04517=1054.030,-84.471,433.269,170.530,29.298,155.538
C04518=1054.024,-84.720,433.280,170.527,29.297,155.538
C04519=1054.018,-84.970,433.291,170.525,29.296,155.538
C04520=1054.012,-85.220,433.302,170.523,29.295,155.537
C04521=1054.005,-85.470,433.313,170.522,29.294,155.537
C04522=1054.000,-85.719,433.324,170.520,29.293,155.537
C04523=1053.994,-85.969,433.335,170.518,29.292,155.537
C04524=1053.987,-86.218,433.345,170.516,29.291,155.537
C04525=1053.981,-86.468,433.356,170.514,29.290,155.537
C04526=1053.975,-86.718,433.367,170.511,29.288,155.537
C04527=1053.968,-86.967,433.378,170.510,29.287,155.537
C04528=1053.962,-87.217,433.389,170.508,29.286,155.537
C04529=1053.956,-87.467,433.400,170.506,29.285,155.537
C04530=1053.950,-87.716,433.410,170.504,29.284,155.537
C04531=1053.944,-87.966,433.421,170.502,29.283,155.537
C04532=1053.938,-88.216,433.432,170.500,29.282,155.537
C04533=1053.931,-88.465,433.443,170.497,29.281,155.537
C04534=1053.926,-88.715,433.453,170.496,29.280,155.537
C04535=1053.919,-88.965,433.464,170.494,29.279,155.537
C04536=1053.913,-89.214,433.474,170.492,29.278,155.537
C04537=1053.907,-89.464,433.485,170.490,29.277,155.537
C04538=1053.901,-89.714,433.496,170.488,29.276,155.537
C04539=1053.894,-89.963,433.507,170.486,29.275,155.537
C04540=1053.888,-90.213,433.518,170.484,29.274,155.537
C04541=1053.882,-90.464,433.528,170.482,29.272,155.537
C04542=1053.876,-90.713,433.538,170.480,29.271,155.537
C04543=1053.870,-90.962,433.549,170.478,29.270,155.537
C04544=1053.863,-91.212,433.560,170.476,29.269,155.537
C04545=1053.857,-91.462,433.571,170.474,29.268,155.537
C04546=1053.852,-91.711,433.582,170.472,29.267,155.537
C04547=1053.845,-91.961,433.591,170.471,29.266,155.537
C04548=1053.839,-92.211,433.602,170.469,29.265,155.536
C04549=1053.833,-92.461,433.613,170.466,29.264,155.536
C04550=1053.827,-92.710,433.624,170.464,29.263,155.536
C04551=1053.822,-92.960,433.634,170.462,29.263,155.537
C04552=1053.814,-93.210,433.644,170.460,29.262,155.537
C04553=1053.809,-93.459,433.655,170.458,29.261,155.536
C04554=1053.803,-93.709,433.666,170.456,29.260,155.536
C04555=1053.797,-93.959,433.676,170.455,29.259,155.536
C04556=1053.790,-94.209,433.687,170.452,29.257,155.536
C04557=1053.785,-94.458,433.698,170.450,29.256,155.536
C04558=1053.778,-94.707,433.708,170.448,29.255,155.536
C04559=1053.773,-94.958,433.718,170.446,29.254,155.536
C04560=1053.766,-95.207,433.729,170.444,29.253,155.536
C04561=1053.760,-95.457,433.740,170.443,29.252,155.536
C04562=1053.754,-95.707,433.749,170.441,29.252,155.536
C04563=1053.748,-95.956,433.760,170.438,29.251,155.536
C04564=1053.742,-96.206,433.771,170.436,29.250,155.536
C04565=1053.736,-96.455,433.781,170.434,29.249,155.536
C04566=1053.730,-96.706,433.792,170.432,29.248,155.536
C04567=1053.723,-96.955,433.802,170.430,29.247,155.536
C04568=1053.718,-97.205,433.812,170.429,29.246,155.536
C04569=1053.712,-97.454,433.823,170.427,29.245,155.536
C04570=1053.706,-97.704,433.833,170.425,29.244,155.536
C04571=1053.699,-97.954,433.843,170.422,29.243,155.536
C04572=1053.693,-98.204,433.854,170.420,29.242,155.536
C04573=1053.687,-98.453,433.864,170.418,29.242,155.536
C04574=1053.680,-98.739,433.876,170.416,29.241,155.536
C04575=1053.673,-99.025,433.888,170.414,29.239,155.536
C04576=1053.666,-99.311,433.899,170.412,29.238,155.536
C04577=1053.659,-99.597,433.911,170.409,29.238,155.536
C04578=1053.652,-99.847,433.921,170.407,29.237,155.536
C04579=1053.647,-100.096,433.931,170.405,29.236,155.536
C04580=1053.640,-100.345,433.942,170.403,29.235,155.536
C04581=1053.633,-100.596,433.952,170.401,29.234,155.536
C04582=1053.628,-100.846,433.962,170.398,29.233,155.536
C04583=1053.622,-101.095,433.972,170.397,29.233,155.536
C04584=1053.615,-101.345,433.982,170.395,29.232,155.536
C04585=1053.610,-101.594,433.993,170.393,29.231,155.536
C04586=1053.603,-101.844,434.002,170.391,29.230,155.536
C04587=1053.596,-102.094,434.013,170.389,29.229,155.536
C04588=1053.591,-102.344,434.023,170.386,29.229,155.536
C04589=1053.584,-102.593,434.033,170.384,29.228,155.536
C04590=1053.578,-102.843,434.043,170.383,29.227,155.536
C04591=1053.573,-103.093,434.054,170.381,29.226,155.536
C04592=1053.566,-103.342,434.063,170.379,29.225,155.536
C04593=1053.560,-103.592,434.073,170.377,29.225,155.536
C04594=1053.554,-103.842,434.084,170.375,29.224,155.536
C04595=1053.548,-104.091,434.093,170.372,29.223,155.536
C04596=1053.541,-104.341,434.104,170.370,29.222,155.537
C04597=1053.535,-104.591,434.113,170.368,29.221,155.536
C04598=1053.530,-104.841,434.124,170.366,29.221,155.537
C04599=1053.523,-105.090,434.134,170.365,29.220,155.537
C04600=1053.517,-105.340,434.143,170.363,29.219,155.537
C04601=1053.512,-105.590,434.154,170.360,29.218,155.537
C04602=1053.505,-105.839,434.164,170.358,29.218,155.537
C04603=1053.499,-106.089,434.173,170.356,29.217,155.537
C04604=1053.493,-106.339,434.183,170.354,29.216,155.537
C04605=1053.487,-106.589,434.194,170.352,29.215,155.537
C04606=1053.481,-106.838,434.203,170.350,29.215,155.537
C04607=1053.475,-107.088,434.213,170.348,29.214,155.537
C04608=1053.468,-107.337,434.223,170.346,29.213,155.537
C04609=1053.462,-107.587,434.233,170.344,29.212,155.537
C04610=1053.456,-107.838,434.243,170.342,29.212,155.537
C04611=1053.450,-108.088,434.253,170.340,29.212,155.537
C04612=1053.443,-108.337,434.263,170.338,29.211,155.537
C04613=1053.437,-108.587,434.273,170.335,29.210,155.537
C04614=1053.431,-108.837,434.282,170.333,29.209,155.537
C04615=1053.425,-109.086,434.292,170.331,29.208,155.537
C04616=1053.419,-109.336,434.302,170.330,29.208,155.537
C04617=1053.412,-109.585,434.312,170.328,29.207,155.537
C04618=1053.407,-109.835,434.322,170.326,29.207,155.537
C04619=1053.401,-110.085,434.332,170.323,29.206,155.537
C04620=1053.394,-110.335,434.341,170.321,29.205,155.537
C04621=1053.388,-110.585,434.351,170.319,29.205,155.537
C04622=1053.382,-110.834,434.361,170.317,29.204,155.537
C04623=1053.376,-111.084,434.371,170.315,29.203,155.537
C04624=1053.369,-111.334,434.380,170.313,29.203,155.538
C04625=1053.363,-111.583,434.390,170.311,29.202,155.538
C04626=1053.357,-111.833,434.399,170.309,29.201,155.538
C04627=1053.351,-112.083,434.409,170.307,29.201,155.538
C04628=1053.345,-112.333,434.419,170.305,29.200,155.538
C04629=1053.339,-112.582,434.429,170.303,29.199,155.538
C04630=1053.333,-112.832,434.439,170.301,29.199,155.538
C04631=1053.327,-113.082,434.448,170.298,29.198,155.538
C04632=1053.320,-113.332,434.458,170.296,29.197,155.538
C04633=1053.314,-113.581,434.468,170.294,29.197,155.538
C04634=1053.308,-113.831,434.477,170.293,29.197,155.538
C04635=1053.302,-114.081,434.487,170.291,29.196,155.538
C04636=1053.296,-114.330,434.496,170.289,29.195,155.538
C04637=1053.290,-114.580,434.505,170.286,29.195,155.538
C04638=1053.283,-114.864,434.517,170.284,29.194,155.538
C04639=1053.276,-115.149,434.527,170.281,29.194,155.538
C04640=1053.269,-115.433,434.538,170.279,29.193,155.538
C04641=1053.262,-115.718,434.550,170.276,29.192,155.538
C04642=1053.255,-115.968,434.559,170.274,29.192,155.539
C04643=1053.249,-116.217,434.568,170.273,29.191,155.539
C04644=1053.243,-116.467,434.578,170.271,29.191,155.539
C04645=1053.237,-116.717,434.587,170.269,29.190,155.539
C04646=1053.231,-116.967,434.597,170.267,29.190,155.539
C04647=1053.224,-117.217,434.606,170.264,29.189,155.539
C04648=1053.219,-117.466,434.616,170.262,29.188,155.539
C04649=1053.213,-117.715,434.625,170.260,29.188,155.539
C04650=1053.207,-117.965,434.635,170.258,29.187,155.539
C04651=1053.200,-118.215,434.644,170.256,29.187,155.539
C04652=1053.194,-118.465,434.654,170.253,29.186,155.539
C04653=1053.188,-118.715,434.663,170.251,29.186,155.539
C04654=1053.182,-118.965,434.672,170.250,29.186,155.539
C04655=1053.176,-119.215,434.682,170.248,29.185,155.540
C04656=1053.170,-119.465,434.691,170.246,29.185,155.540
C04657=1053.164,-119.713,434.700,170.244,29.184,155.540
C04658=1053.157,-119.963,434.710,170.241,29.184,155.540
C04659=1053.151,-120.213,434.719,170.239,29.183,155.540
C04660=1053.145,-120.463,434.729,170.237,29.183,155.540
C04661=1053.139,-120.713,434.738,170.235,29.182,155.540
C04662=1053.133,-120.963,434.747,170.233,29.182,155.540
C04663=1053.127,-121.213,434.757,170.230,29.181,155.540
C04664=1053.121,-121.462,434.766,170.229,29.181,155.540
C04665=1053.114,-121.711,434.775,170.227,29.180,155.540
C04666=1053.108,-121.961,434.784,170.225,29.180,155.540
C04667=1053.102,-122.212,434.793,170.223,29.179,155.540
C04668=1053.096,-122.461,434.803,170.221,29.180,155.541
C04669=1053.091,-122.711,434.812,170.218,29.179,155.541
C04670=1053.084,-122.960,434.822,170.216,29.179,155.541
C04671=1053.077,-123.210,434.831,170.214,29.178,155.541
C04672=1053.072,-123.460,434.839,170.212,29.178,155.541
C04673=1053.065,-123.710,434.849,170.210,29.177,155.541
C04674=1053.059,-123.960,434.859,170.207,29.177,155.541
C04675=1053.054,-124.210,434.867,170.205,29.176,155.541
C04676=1053.048,-124.459,434.877,170.203,29.176,155.541
C04677=1053.041,-124.709,434.886,170.202,29.176,155.541
C04678=1053.035,-124.959,434.895,170.200,29.175,155.542
C04679=1053.029,-125.209,434.904,170.198,29.175,155.542
C04680=1053.023,-125.458,434.913,170.195,29.175,155.542
C04681=1053.016,-125.708,434.922,170.193,29.174,155.542
C04682=1053.011,-125.958,434.931,170.191,29.174,155.542
C04683=1053.004,-126.208,434.941,170.189,29.174,155.542
C04684=1052.998,-126.457,434.949,170.187,29.173,155.542
C04685=1052.992,-126.707,434.958,170.184,29.173,155.542
C04686=1052.986,-126.957,434.968,170.182,29.173,155.542
C04687=1052.979,-127.206,434.977,170.180,29.172,155.543
C04688=1052.974,-127.456,434.985,170.178,29.172,155.543
C04689=1052.968,-127.706,434.995,170.176,29.172,155.543
C04690=1052.962,-127.956,435.004,170.174,29.171,155.543
C04691=1052.958,-128.206,435.014,170.172,29.170,155.543
C04692=1052.954,-128.456,435.024,170.170,29.168,155.543
C04693=1052.952,-128.705,435.035,170.169,29.167,155.542
C04694=1052.950,-128.956,435.048,170.168,29.164,155.542
C04695=1052.950,-129.207,435.060,170.166,29.161,155.542
C04696=1052.952,-129.457,435.073,170.164,29.157,155.541
C04697=1052.954,-129.707,435.088,170.164,29.153,155.541
C04698=1052.957,-129.958,435.102,170.162,29.149,155.540
C04699=1052.961,-130.210,435.118,170.162,29.143,155.539
C04700=1052.968,-130.460,435.133,170.162,29.138,155.538
C04701=1052.974,-130.710,435.149,170.160,29.132,155.537
C04702=1052.605,-130.733,434.933,170.113,29.300,155.570
C04703=1052.599,-130.483,434.917,170.115,29.306,155.571
C04704=1052.593,-130.233,434.900,170.115,29.312,155.572
C04705=1052.588,-129.982,434.885,170.116,29.317,155.573
C04706=1052.585,-129.731,434.870,170.117,29.322,155.573
C04707=1052.583,-129.481,434.857,170.118,29.325,155.574
C04708=1052.582,-129.230,434.843,170.119,29.329,155.574
C04709=1052.581,-128.980,434.830,170.120,29.332,155.575
C04710=1052.583,-128.729,434.818,170.122,29.334,155.575
C04711=1052.585,-128.480,434.807,170.123,29.337,155.575
C04712=1052.588,-128.229,434.797,170.125,29.338,155.576
C04713=1052.592,-127.979,434.786,170.127,29.339,155.576
C04714=1052.599,-127.729,434.777,170.129,29.340,155.576
C04715=1052.604,-127.479,434.768,170.132,29.340,155.575
C04716=1052.611,-127.230,434.759,170.134,29.341,155.575
C04717=1052.617,-126.980,434.750,170.136,29.341,155.575
C04718=1052.623,-126.730,434.741,170.138,29.341,155.575
C04719=1052.630,-126.480,434.732,170.139,29.341,155.575
C04720=1052.635,-126.231,434.723,170.142,29.342,155.575
C04721=1052.641,-125.981,434.714,170.144,29.342,155.575
C04722=1052.647,-125.731,434.704,170.146,29.343,155.575
C04723=1052.654,-125.482,434.695,170.148,29.343,155.575
C04724=1052.659,-125.232,434.687,170.150,29.343,155.574
C04725=1052.666,-124.982,434.677,170.153,29.343,155.574
C04726=1052.673,-124.733,434.668,170.155,29.344,155.574
C04727=1052.678,-124.482,434.660,170.157,29.344,155.574
C04728=1052.685,-124.232,434.650,170.159,29.345,155.574
C04729=1052.690,-123.983,434.641,170.161,29.345,155.574
C04730=1052.696,-123.734,434.631,170.164,29.346,155.574
C04731=1052.703,-123.483,434.623,170.165,29.346,155.574
C04732=1052.709,-123.234,434.613,170.167,29.346,155.574
C04733=1052.715,-122.984,434.604,170.169,29.347,155.574
C04734=1052.721,-122.735,434.595,170.171,29.347,155.573
C04735=1052.727,-122.484,434.586,170.173,29.347,155.573
C04736=1052.733,-122.235,434.576,170.176,29.347,155.573
C04737=1052.740,-121.985,434.567,170.178,29.348,155.573
C04738=1052.746,-121.735,434.558,170.180,29.348,155.573
C04739=1052.752,-121.485,434.548,170.182,29.349,155.573
C04740=1052.757,-121.236,434.540,170.184,29.349,155.573
C04741=1052.764,-120.986,434.530,170.187,29.350,155.573
C04742=1052.770,-120.736,434.520,170.189,29.350,155.573
C04743=1052.776,-120.486,434.511,170.190,29.350,155.573
C04744=1052.783,-120.237,434.502,170.192,29.351,155.573
C04745=1052.789,-119.987,434.492,170.194,29.351,155.573
C04746=1052.795,-119.737,434.483,170.197,29.352,155.572
C04747=1052.800,-119.488,434.474,170.199,29.353,155.572
C04748=1052.807,-119.238,434.465,170.201,29.353,155.572
C04749=1052.813,-118.988,434.455,170.203,29.354,155.572
C04750=1052.819,-118.738,434.446,170.205,29.354,155.572
C04751=1052.825,-118.488,434.436,170.207,29.354,155.572
C04752=1052.831,-118.239,434.426,170.210,29.355,155.572
C04753=1052.837,-117.989,434.417,170.212,29.355,155.572
C04754=1052.844,-117.739,434.408,170.213,29.356,155.572
C04755=1052.850,-117.490,434.399,170.215,29.356,155.572
C04756=1052.856,-117.240,434.389,170.217,29.357,155.572
C04757=1052.862,-116.991,434.380,170.220,29.357,155.572
C04758=1052.868,-116.741,434.370,170.222,29.358,155.572
C04759=1052.875,-116.491,434.360,170.224,29.359,155.572
C04760=1052.881,-116.241,434.351,170.226,29.359,155.571
C04761=1052.887,-115.991,434.341,170.228,29.359,155.571
C04762=1052.893,-115.742,434.332,170.231,29.360,155.571
C04763=1052.900,-115.457,434.321,170.233,29.360,155.571
C04764=1052.907,-115.172,434.311,170.235,29.361,155.571
C04765=1052.914,-114.888,434.300,170.237,29.362,155.571
C04766=1052.921,-114.603,434.288,170.239,29.362,155.571
C04767=1052.927,-114.353,434.279,170.242,29.363,155.571
C04768=1052.933,-114.103,434.269,170.244,29.363,155.571
C04769=1052.939,-113.853,434.260,170.246,29.364,155.571
C04770=1052.945,-113.604,434.250,170.248,29.365,155.571
C04771=1052.951,-113.355,434.241,170.250,29.365,155.571
C04772=1052.957,-113.105,434.231,170.253,29.366,155.571
C04773=1052.964,-112.856,434.221,170.255,29.367,155.571
C04774=1052.970,-112.606,434.211,170.256,29.367,155.571
C04775=1052.976,-112.356,434.202,170.258,29.367,155.571
C04776=1052.982,-112.106,434.192,170.260,29.368,155.570
C04777=1052.988,-111.856,434.183,170.262,29.369,155.570
C04778=1052.995,-111.607,434.173,170.265,29.369,155.570
C04779=1053.000,-111.356,434.163,170.267,29.370,155.570
C04780=1053.006,-111.107,434.153,170.269,29.371,155.570
C04781=1053.013,-110.857,434.143,170.271,29.371,155.570
C04782=1053.019,-110.608,434.134,170.273,29.372,155.570
C04783=1053.025,-110.358,434.124,170.276,29.373,155.570
C04784=1053.031,-110.108,434.114,170.277,29.373,155.570
C04785=1053.037,-109.858,434.105,170.279,29.374,155.570
C04786=1053.044,-109.609,434.095,170.281,29.375,155.570
C04787=1053.050,-109.359,434.085,170.283,29.375,155.570
C04788=1053.055,-109.109,434.075,170.285,29.375,155.570
C04789=1053.062,-108.859,434.065,170.288,29.377,155.570
C04790=1053.068,-108.610,434.056,170.290,29.377,155.570
C04791=1053.074,-108.360,434.045,170.292,29.377,155.570
C04792=1053.081,-108.110,434.036,170.294,29.378,155.570
C04793=1053.087,-107.860,434.026,170.295,29.379,155.570
C04794=1053.093,-107.610,434.016,170.297,29.380,155.570
C04795=1053.100,-107.361,434.006,170.300,29.380,155.570
C04796=1053.105,-107.111,433.996,170.302,29.381,155.570
C04797=1053.111,-106.861,433.986,170.304,29.382,155.570
C04798=1053.118,-106.612,433.976,170.306,29.382,155.569
C04799=1053.124,-106.362,433.967,170.308,29.383,155.570
C04800=1053.129,-106.112,433.956,170.310,29.384,155.569
C04801=1053.136,-105.863,433.946,170.313,29.385,155.569
C04802=1053.142,-105.613,433.937,170.314,29.385,155.569
C04803=1053.148,-105.363,433.927,170.316,29.386,155.569
C04804=1053.154,-105.114,433.916,170.318,29.387,155.569
C04805=1053.160,-104.864,433.906,170.320,29.388,155.569
C04806=1053.166,-104.614,433.897,170.322,29.388,155.569
C04807=1053.173,-104.364,433.886,170.325,29.389,155.569
C04808=1053.179,-104.114,433.876,170.327,29.390,155.569
C04809=1053.185,-103.864,433.867,170.329,29.391,155.569
C04810=1053.192,-103.615,433.856,170.330,29.392,155.569
C04811=1053.197,-103.365,433.846,170.332,29.392,155.569
C04812=1053.203,-103.116,433.836,170.334,29.393,155.569
C04813=1053.210,-102.866,433.826,170.337,29.394,155.569
C04814=1053.215,-102.616,433.816,170.339,29.395,155.569
C04815=1053.222,-102.367,433.806,170.341,29.396,155.569
C04816=1053.228,-102.116,433.796,170.343,29.396,155.569
C04817=1053.234,-101.867,433.785,170.345,29.397,155.569
C04818=1053.240,-101.617,433.775,170.347,29.397,155.569
C04819=1053.247,-101.368,433.765,170.349,29.399,155.569
C04820=1053.252,-101.118,433.755,170.351,29.400,155.569
C04821=1053.259,-100.869,433.745,170.353,29.400,155.569
C04822=1053.265,-100.619,433.735,170.355,29.401,155.569
C04823=1053.271,-100.369,433.724,170.357,29.402,155.569
C04824=1053.277,-100.119,433.714,170.359,29.402,155.569
C04825=1053.284,-99.870,433.704,170.362,29.404,155.569
C04826=1053.289,-99.620,433.694,170.364,29.404,155.569
C04827=1053.296,-99.334,433.682,170.365,29.405,155.569
C04828=1053.304,-99.048,433.670,170.368,29.406,155.569
C04829=1053.311,-98.762,433.658,170.370,29.407,155.569
C04830=1053.318,-98.476,433.647,170.373,29.408,155.569
C04831=1053.324,-98.227,433.637,170.375,29.409,155.569
C04832=1053.331,-97.977,433.627,170.377,29.410,155.569
C04833=1053.337,-97.727,433.616,170.379,29.411,155.569
C04834=1053.343,-97.477,433.606,170.380,29.411,155.569
C04835=1053.348,-97.228,433.595,170.382,29.412,155.569
C04836=1053.355,-96.979,433.585,170.384,29.413,155.569
C04837=1053.361,-96.728,433.574,170.387,29.414,155.569
C04838=1053.367,-96.478,433.564,170.389,29.415,155.569
C04839=1053.373,-96.229,433.554,170.391,29.416,155.569
C04840=1053.379,-95.979,433.543,170.393,29.417,155.569
C04841=1053.385,-95.730,433.533,170.395,29.418,155.569
C04842=1053.391,-95.479,433.522,170.396,29.419,155.569
C04843=1053.398,-95.230,433.512,170.398,29.420,155.569
C04844=1053.403,-94.980,433.501,170.401,29.421,155.569
C04845=1053.409,-94.730,433.491,170.403,29.422,155.569
C04846=1053.415,-94.481,433.481,170.405,29.423,155.569
C04847=1053.422,-94.231,433.469,170.407,29.424,155.569
C04848=1053.428,-93.982,433.459,170.409,29.424,155.569
C04849=1053.434,-93.732,433.449,170.410,29.425,155.569
C04850=1053.439,-93.482,433.438,170.412,29.426,155.569
C04851=1053.446,-93.232,433.428,170.415,29.427,155.569
C04852=1053.452,-92.983,433.417,170.417,29.428,155.569
C04853=1053.458,-92.733,433.406,170.419,29.429,155.569
C04854=1053.464,-92.484,433.396,170.421,29.431,155.569
C04855=1053.470,-92.233,433.385,170.423,29.432,155.569
C04856=1053.477,-91.984,433.375,170.424,29.433,155.569
C04857=1053.482,-91.734,433.365,170.426,29.434,155.569
C04858=1053.488,-91.485,433.354,170.429,29.435,155.569
C04859=1053.495,-91.235,433.343,170.431,29.436,155.569
C04860=1053.501,-90.985,433.332,170.433,29.437,155.569
C04861=1053.507,-90.736,433.321,170.435,29.438,155.570
C04862=1053.514,-90.486,433.311,170.437,29.439,155.570
C04863=1053.519,-90.236,433.300,170.438,29.440,155.570
C04864=1053.526,-89.987,433.290,170.440,29.441,155.570
C04865=1053.532,-89.736,433.279,170.443,29.441,155.570
C04866=1053.538,-89.487,433.268,170.445,29.442,155.570
C04867=1053.544,-89.238,433.258,170.447,29.443,155.570
C04868=1053.550,-88.987,433.246,170.449,29.444,155.570
C04869=1053.556,-88.738,433.236,170.451,29.445,155.570
C04870=1053.562,-88.488,433.226,170.452,29.446,155.570
C04871=1053.569,-88.238,433.215,170.454,29.448,155.570
C04872=1053.574,-87.988,433.204,170.456,29.449,155.570
C04873=1053.581,-87.739,433.194,170.459,29.450,155.570
C04874=1053.587,-87.489,433.182,170.461,29.451,155.570
C04875=1053.593,-87.240,433.172,170.463,29.452,155.570
C04876=1053.599,-86.990,433.161,170.464,29.453,155.570
C04877=1053.606,-86.740,433.150,170.466,29.454,155.570
C04878=1053.612,-86.491,433.139,170.468,29.455,155.570
C04879=1053.619,-86.241,433.128,170.470,29.456,155.570
C04880=1053.624,-85.991,433.118,170.473,29.457,155.570
C04881=1053.630,-85.742,433.107,170.475,29.458,155.570
C04882=1053.636,-85.492,433.095,170.477,29.459,155.570
C04883=1053.643,-85.243,433.085,170.478,29.460,155.570
C04884=1053.649,-84.992,433.074,170.480,29.461,155.570
C04885=1053.655,-84.743,433.063,170.482,29.462,155.570
C04886=1053.661,-84.494,433.053,170.484,29.463,155.570
C04887=1053.668,-84.244,433.042,170.486,29.464,155.570
C04888=1053.674,-83.994,433.031,170.489,29.465,155.570
C04889=1053.681,-83.744,433.020,170.491,29.467,155.571
C04890=1053.686,-83.495,433.009,170.492,29.468,155.571
C04891=1053.693,-83.211,432.996,170.494,29.469,155.571
C04892=1053.701,-82.928,432.985,170.497,29.470,155.571
C04893=1053.708,-82.644,432.972,170.499,29.471,155.571
C04894=1053.715,-82.360,432.960,170.501,29.473,155.571
C04895=1053.721,-82.111,432.948,170.504,29.474,155.571
C04896=1053.728,-81.861,432.937,170.505,29.475,155.571
C04897=1053.734,-81.611,432.926,170.507,29.476,155.571
C04898=1053.740,-81.361,432.915,170.509,29.477,155.571
C04899=1053.746,-81.112,432.904,170.511,29.478,155.571
C04900=1053.753,-80.862,432.894,170.513,29.480,155.571
C04901=1053.758,-80.612,432.883,170.515,29.481,155.571
C04902=1053.765,-80.362,432.871,170.517,29.482,155.571
C04903=1053.772,-80.114,432.861,170.519,29.483,155.571
C04904=1053.778,-79.863,432.849,170.521,29.484,155.571
C04905=1053.784,-79.614,432.838,170.523,29.485,155.571
C04906=1053.790,-79.364,432.827,170.525,29.486,155.571
C04907=1053.796,-79.114,432.816,170.527,29.487,155.571
C04908=1053.802,-78.865,432.804,170.529,29.488,155.571
C04909=1053.808,-78.615,432.793,170.530,29.490,155.572
C04910=1053.814,-78.365,432.782,170.532,29.491,155.572
C04911=1053.820,-78.115,432.771,170.534,29.492,155.572
C04912=1053.827,-77.866,432.759,170.537,29.494,155.572
C04913=1053.833,-77.616,432.748,170.539,29.495,155.572
C04914=1053.839,-77.366,432.737,170.541,29.496,155.572
C04915=1053.845,-77.117,432.726,170.542,29.497,155.572
C04916=1053.851,-76.867,432.714,170.544,29.498,155.572
C04917=1053.857,-76.618,432.704,170.546,29.499,155.572
C04918=1053.863,-76.367,432.692,170.548,29.501,155.572
C04919=1053.869,-76.118,432.681,170.550,29.502,155.572
C04920=1053.876,-75.868,432.669,170.552,29.504,155.572
C04921=1053.882,-75.619,432.659,170.553,29.505,155.573
C04922=1053.889,-75.369,432.648,170.556,29.506,155.573
C04923=1053.895,-75.120,432.636,170.558,29.507,155.573
C04924=1053.901,-74.870,432.625,170.560,29.508,155.573
C04925=1053.907,-74.620,432.614,170.562,29.509,155.573
C04926=1053.913,-74.371,432.602,170.564,29.511,155.573
C04927=1053.920,-74.121,432.591,170.565,29.512,155.573
C04928=1053.926,-73.872,432.579,170.567,29.514,155.573
C04929=1053.931,-73.621,432.568,170.569,29.515,155.573
C04930=1053.937,-73.372,432.557,170.571,29.516,155.573
C04931=1053.944,-73.122,432.545,170.573,29.517,155.573
C04932=1053.949,-72.873,432.534,170.575,29.519,155.573
C04933=1053.955,-72.623,432.521,170.577,29.521,155.574
C04934=1053.961,-72.373,432.510,170.579,29.522,155.574
C04935=1053.968,-72.124,432.498,170.581,29.523,155.574
C04936=1053.974,-71.874,432.487,170.583,29.524,155.574
C04937=1053.980,-71.624,432.476,170.585,29.526,155.574
C04938=1053.986,-71.374,432.464,170.587,29.527,155.574
C04939=1053.991,-71.125,432.453,170.588,29.528,155.574
C04940=1053.998,-70.875,432.441,170.590,29.530,155.574
C04941=1054.004,-70.626,432.430,170.592,29.531,155.574
C04942=1054.010,-70.376,432.418,170.594,29.533,155.574
C04943=1054.015,-70.126,432.407,170.596,29.534,155.575
C04944=1054.022,-69.877,432.395,170.597,29.535,155.575
C04945=1054.029,-69.627,432.383,170.599,29.537,155.575
C04946=1054.034,-69.377,432.371,170.602,29.538,155.575
C04947=1054.040,-69.128,432.359,170.604,29.540,155.575
C04948=1054.046,-68.878,432.348,170.606,29.541,155.575
C04949=1054.053,-68.629,432.336,170.608,29.542,155.575
C04950=1054.058,-68.378,432.325,170.609,29.544,155.575
C04951=1054.064,-68.129,432.313,170.611,29.545,155.575
C04952=1054.071,-67.879,432.302,170.613,29.546,155.576
C04953=1054.077,-67.630,432.290,170.615,29.548,155.576
C04954=1054.083,-67.380,432.278,170.617,29.549,155.576
C04955=1054.090,-67.099,432.265,170.619,29.551,155.576
C04956=1054.097,-66.817,432.251,170.621,29.552,155.576
C04957=1054.103,-66.536,432.238,170.623,29.554,155.576
C04958=1054.111,-66.255,432.225,170.625,29.556,155.576
C04959=1054.116,-66.005,432.213,170.628,29.557,155.576
C04960=1054.123,-65.755,432.201,170.630,29.558,155.576
C04961=1054.129,-65.506,432.190,170.631,29.560,155.577
C04962=1054.135,-65.256,432.178,170.633,29.562,155.577
C04963=1054.141,-65.006,432.166,170.635,29.563,155.577
C04964=1054.147,-64.757,432.154,170.637,29.564,155.577
C04965=1054.154,-64.507,432.143,170.639,29.566,155.577
C04966=1054.159,-64.257,432.130,170.640,29.567,155.577
C04967=1054.166,-64.008,432.119,170.642,29.568,155.577
C04968=1054.172,-63.758,432.108,170.644,29.570,155.577
C04969=1054.178,-63.508,432.095,170.646,29.572,155.578
C04970=1054.184,-63.259,432.083,170.648,29.573,155.578
C04971=1054.190,-63.010,432.072,170.650,29.574,155.578
C04972=1054.196,-62.759,432.060,170.651,29.576,155.578
C04973=1054.203,-62.510,432.048,170.653,29.577,155.578
C04974=1054.209,-62.260,432.036,170.655,29.578,155.578
C04975=1054.215,-62.011,432.024,170.658,29.580,155.578
C04976=1054.221,-61.761,432.012,170.660,29.582,155.578
C04977=1054.228,-61.511,432.000,170.661,29.583,155.579
C04978=1054.234,-61.261,431.988,170.663,29.584,155.579
C04979=1054.240,-61.012,431.976,170.665,29.586,155.579
C04980=1054.246,-60.763,431.964,170.667,29.588,155.579
C04981=1054.252,-60.513,431.952,170.669,29.589,155.579
C04982=1054.259,-60.263,431.940,170.671,29.590,155.579
C04983=1054.265,-60.013,431.929,170.672,29.592,155.579
C04984=1054.270,-59.764,431.916,170.674,29.593,155.579
C04985=1054.277,-59.514,431.904,170.676,29.595,155.580
C04986=1054.284,-59.265,431.892,170.678,29.596,155.580
C04987=1054.290,-59.015,431.880,170.680,29.598,155.580
C04988=1054.296,-58.765,431.869,170.681,29.599,155.580
C04989=1054.302,-58.516,431.857,170.683,29.601,155.580
C04990=1054.308,-58.266,431.844,170.685,29.602,155.580
C04991=1054.315,-58.016,431.833,170.687,29.603,155.580
C04992=1054.321,-57.767,431.821,170.689,29.605,155.580
C04993=1054.327,-57.517,431.808,170.691,29.607,155.581
C04994=1054.334,-57.267,431.796,170.693,29.608,155.581
C04995=1054.339,-57.018,431.784,170.695,29.610,155.581
C04996=1054.346,-56.769,431.772,170.697,29.611,155.581
C04997=1054.352,-56.519,431.760,170.699,29.613,155.581
C04998=1054.358,-56.269,431.747,170.701,29.614,155.581
C04999=1054.365,-56.020,431.735,170.702,29.616,155.581
C05000=1054.372,-55.770,431.723,170.704,29.617,155.581
C05001=1054.378,-55.520,431.711,170.706,29.619,155.582
C05002=1054.384,-55.271,431.699,170.708,29.620,155.582
C05003=1054.389,-55.021,431.687,170.710,29.621,155.582
C05004=1054.396,-54.772,431.675,170.711,29.623,155.582
C05005=1054.403,-54.522,431.663,170.713,29.625,155.582
C05006=1054.409,-54.272,431.650,170.715,29.626,155.582
C05007=1054.415,-54.023,431.638,170.717,29.628,155.582
C05008=1054.421,-53.773,431.626,170.719,29.629,155.583
C05009=1054.428,-53.523,431.614,170.721,29.630,155.583
C05010=1054.434,-53.273,431.601,170.722,29.632,155.583
C05011=1054.440,-53.024,431.589,170.724,29.634,155.583
C05012=1054.447,-52.774,431.577,170.726,29.635,155.583
C05013=1054.453,-52.524,431.565,170.728,29.637,155.583
C05014=1054.460,-52.275,431.553,170.730,29.638,155.583
C05015=1054.466,-52.025,431.540,170.731,29.640,155.584
C05016=1054.472,-51.776,431.529,170.733,29.641,155.584
C05017=1054.478,-51.527,431.517,170.735,29.643,155.584
C05018=1054.484,-51.277,431.504,170.738,29.644,155.584
C05019=1054.492,-50.997,431.490,170.740,29.646,155.584
C05020=1054.499,-50.716,431.476,170.741,29.648,155.584
C05021=1054.506,-50.436,431.462,170.743,29.650,155.584
C05022=1054.513,-50.156,431.448,170.746,29.652,155.585
C05023=1054.519,-49.907,431.436,170.748,29.653,155.585
C05024=1054.525,-49.657,431.424,170.750,29.655,155.585
C05025=1054.531,-49.407,431.411,170.751,29.656,155.585
C05026=1054.537,-49.157,431.398,170.753,29.658,155.585
C05027=1054.544,-48.908,431.386,170.755,29.660,155.585
C05028=1054.550,-48.658,431.373,170.757,29.662,155.586
C05029=1054.556,-48.408,431.361,170.759,29.663,155.586
C05030=1054.562,-48.159,431.348,170.760,29.665,155.586
C05031=1054.569,-47.910,431.335,170.762,29.666,155.586
C05032=1054.574,-47.660,431.323,170.764,29.668,155.586
C05033=1054.580,-47.411,431.311,170.766,29.670,155.586
C05034=1054.586,-47.161,431.298,170.768,29.671,155.587
C05035=1054.593,-46.912,431.285,170.769,29.673,155.587
C05036=1054.599,-46.662,431.273,170.771,29.675,155.587
C05037=1054.605,-46.412,431.260,170.773,29.677,155.587
C05038=1054.611,-46.163,431.247,170.775,29.678,155.587
C05039=1054.617,-45.913,431.235,170.777,29.680,155.587
C05040=1054.623,-45.663,431.223,170.778,29.681,155.588
C05041=1054.630,-45.414,431.209,170.780,29.683,155.588
C05042=1054.635,-45.164,431.197,170.782,29.685,155.588
C05043=1054.641,-44.914,431.184,170.784,29.687,155.588
C05044=1054.648,-44.665,431.172,170.786,29.688,155.588
C05045=1054.654,-44.415,431.159,170.787,29.690,155.588
C05046=1054.660,-44.165,431.146,170.789,29.692,155.589
C05047=1054.666,-43.916,431.133,170.791,29.693,155.589
C05048=1054.672,-43.666,431.121,170.793,29.695,155.589
C05049=1054.679,-43.417,431.109,170.795,29.697,155.589
C05050=1054.685,-43.168,431.095,170.796,29.699,155.589
C05051=1054.691,-42.918,431.083,170.798,29.700,155.590
C05052=1054.697,-42.668,431.070,170.800,29.702,155.590
C05053=1054.704,-42.419,431.058,170.802,29.704,155.590
C05054=1054.711,-42.169,431.044,170.804,29.705,155.590
C05055=1054.717,-41.919,431.031,170.805,29.707,155.590
C05056=1054.723,-41.669,431.019,170.807,29.709,155.590
C05057=1054.729,-41.420,431.006,170.809,29.710,155.591
C05058=1054.735,-41.170,430.993,170.811,29.712,155.591
C05059=1054.742,-40.921,430.980,170.813,29.714,155.591
C05060=1054.747,-40.671,430.968,170.814,29.716,155.591
C05061=1054.754,-40.422,430.955,170.816,29.717,155.591
C05062=1054.760,-40.172,430.942,170.818,29.719,155.591
C05063=1054.766,-39.923,430.929,170.820,29.721,155.592
C05064=1054.772,-39.673,430.917,170.822,29.723,155.592
C05065=1054.779,-39.424,430.903,170.823,29.724,155.592
C05066=1054.785,-39.173,430.891,170.825,29.726,155.592
C05067=1054.791,-38.924,430.877,170.827,29.728,155.592
C05068=1054.797,-38.674,430.865,170.829,29.730,155.593
C05069=1054.804,-38.425,430.851,170.830,29.731,155.593
C05070=1054.809,-38.175,430.839,170.831,29.733,155.593
C05071=1054.816,-37.926,430.826,170.833,29.735,155.593
C05072=1054.822,-37.676,430.812,170.835,29.736,155.593
C05073=1054.828,-37.427,430.800,170.837,29.738,155.594
C05074=1054.834,-37.177,430.787,170.839,29.740,155.594
C05075=1054.840,-36.927,430.774,170.840,29.742,155.594
C05076=1054.847,-36.677,430.760,170.842,29.744,155.594
C05077=1054.853,-36.428,430.747,170.844,29.745,155.594
C05078=1054.859,-36.178,430.735,170.846,29.748,155.595
C05079=1054.865,-35.929,430.721,170.848,29.749,155.595
C05080=1054.871,-35.680,430.708,170.849,29.751,155.595
C05081=1054.877,-35.430,430.695,170.851,29.753,155.595
C05082=1054.883,-35.181,430.682,170.853,29.755,155.595
C05083=1054.890,-34.901,430.667,170.855,29.757,155.596
C05084=1054.898,-34.620,430.653,170.856,29.759,155.596
C05085=1054.904,-34.341,430.638,170.859,29.761,155.596
C05086=1054.911,-34.062,430.623,170.861,29.763,155.596
C05087=1054.917,-33.812,430.610,170.863,29.764,155.597
C05088=1054.923,-33.562,430.597,170.865,29.767,155.597
C05089=1054.929,-33.313,430.583,170.866,29.768,155.597
C05090=1054.935,-33.063,430.570,170.868,29.770,155.597
C05091=1054.942,-32.813,430.557,170.870,29.772,155.597
C05092=1054.948,-32.564,430.544,170.872,29.774,155.598
C05093=1054.954,-32.315,430.530,170.873,29.776,155.598
C05094=1054.960,-32.065,430.517,170.874,29.777,155.598
C05095=1054.966,-31.815,430.504,170.876,29.779,155.598
C05096=1054.973,-31.565,430.491,170.878,29.781,155.598
C05097=1054.979,-31.316,430.478,170.880,29.783,155.599
C05098=1054.985,-31.067,430.464,170.882,29.785,155.599
C05099=1054.991,-30.817,430.452,170.883,29.787,155.599
C05100=1054.997,-30.567,430.437,170.885,29.788,155.599
C05101=1055.004,-30.317,430.424,170.887,29.790,155.599
C05102=1055.010,-30.068,430.411,170.889,29.792,155.600
C05103=1055.016,-29.819,430.398,170.891,29.794,155.600
C05104=1055.022,-29.570,430.384,170.892,29.796,155.600
C05105=1055.029,-29.319,430.371,170.894,29.798,155.600
C05106=1055.035,-29.070,430.358,170.896,29.800,155.601
C05107=1055.041,-28.821,430.345,170.898,29.801,155.601
C05108=1055.048,-28.571,430.331,170.899,29.804,155.601
C05109=1055.054,-28.321,430.317,170.901,29.805,155.601
C05110=1055.060,-28.072,430.304,170.903,29.807,155.601
C05111=1055.066,-27.822,430.291,170.905,29.809,155.602
C05112=1055.073,-27.573,430.277,170.906,29.810,155.602
C05113=1055.079,-27.323,430.264,170.907,29.812,155.602
C05114=1055.085,-27.074,430.251,170.909,29.814,155.602
C05115=1055.092,-26.823,430.238,170.911,29.816,155.602
C05116=1055.097,-26.574,430.224,170.913,29.818,155.603
C05117=1055.103,-26.325,430.211,170.915,29.820,155.603
C05118=1055.110,-26.075,430.197,170.916,29.822,155.603
C05119=1055.116,-25.825,430.183,170.918,29.824,155.603
C05120=1055.122,-25.576,430.170,170.920,29.826,155.604
C05121=1055.127,-25.326,430.156,170.922,29.828,155.604
C05122=1055.134,-25.077,430.143,170.924,29.830,155.604
C05123=1055.140,-24.827,430.129,170.925,29.832,155.604
C05124=1055.146,-24.577,430.115,170.927,29.833,155.604
C05125=1055.152,-24.328,430.102,170.929,29.836,155.605
C05126=1055.159,-24.078,430.088,170.930,29.838,155.605
C05127=1055.164,-23.829,430.075,170.932,29.839,155.605
C05128=1055.171,-23.580,430.061,170.933,29.841,155.605
C05129=1055.177,-23.331,430.047,170.935,29.844,155.606
C05130=1055.183,-23.080,430.033,170.937,29.845,155.606
C05131=1055.189,-22.831,430.020,170.939,29.847,155.606
C05132=1055.195,-22.582,430.006,170.940,29.850,155.606
C05133=1055.202,-22.332,429.992,170.942,29.851,155.607
C05134=1055.208,-22.082,429.979,170.944,29.853,155.607
C05135=1055.213,-21.833,429.965,170.946,29.855,155.607
C05136=1055.220,-21.583,429.951,170.948,29.857,155.607
C05137=1055.226,-21.334,429.938,170.948,29.859,155.608
C05138=1055.232,-21.084,429.924,170.950,29.861,155.608
C05139=1055.239,-20.835,429.910,170.952,29.863,155.608
C05140=1055.245,-20.585,429.896,170.954,29.865,155.608
C05141=1055.251,-20.336,429.883,170.956,29.867,155.609
C05142=1055.258,-20.086,429.869,170.957,29.869,155.609
C05143=1055.263,-19.836,429.855,170.959,29.871,155.609
C05144=1055.270,-19.586,429.842,170.961,29.872,155.609
C05145=1055.276,-19.337,429.827,170.963,29.875,155.609
C05146=1055.282,-19.088,429.814,170.964,29.877,155.610
C05147=1055.289,-18.807,429.798,170.966,29.879,155.610
C05148=1055.296,-18.527,429.783,170.968,29.881,155.610
C05149=1055.303,-18.246,429.767,170.970,29.883,155.611
C05150=1055.309,-17.966,429.752,170.971,29.886,155.611
C05151=1055.316,-17.716,429.738,170.973,29.887,155.611
C05152=1055.322,-17.467,429.725,170.975,29.889,155.611
C05153=1055.329,-17.217,429.710,170.977,29.891,155.612
C05154=1055.335,-16.968,429.696,170.979,29.893,155.612
C05155=1055.341,-16.718,429.682,170.980,29.895,155.612
C05156=1055.347,-16.468,429.669,170.982,29.897,155.612
C05157=1055.353,-16.219,429.654,170.984,29.900,155.613
C05158=1055.360,-15.969,429.641,170.985,29.901,155.613
C05159=1055.366,-15.720,429.627,170.987,29.903,155.613
C05160=1055.373,-15.470,429.612,170.988,29.905,155.613
C05161=1055.379,-15.221,429.599,170.990,29.907,155.613
C05162=1055.385,-14.971,429.585,170.992,29.909,155.614
C05163=1055.391,-14.722,429.571,170.994,29.911,155.614
C05164=1055.397,-14.472,429.557,170.995,29.913,155.614
C05165=1055.403,-14.222,429.543,170.997,29.916,155.615
C05166=1055.409,-13.974,429.529,170.998,29.917,155.615
C05167=1055.415,-13.723,429.515,171.000,29.919,155.615
C05168=1055.421,-13.474,429.501,171.002,29.921,155.615
C05169=1055.428,-13.225,429.486,171.003,29.924,155.616
C05170=1055.434,-12.975,429.473,171.005,29.926,155.616
C05171=1055.440,-12.725,429.458,171.007,29.928,155.616
C05172=1055.446,-12.476,429.444,171.009,29.929,155.616
C05173=1055.453,-12.226,429.429,171.011,29.932,155.617
C05174=1055.458,-11.977,429.416,171.012,29.934,155.617
C05175=1055.464,-11.728,429.402,171.013,29.936,155.617
C05176=1055.471,-11.478,429.387,171.015,29.938,155.617
C05177=1055.476,-11.228,429.374,171.017,29.940,155.618
C05178=1055.483,-10.979,429.359,171.018,29.942,155.618
C05179=1055.489,-10.729,429.345,171.020,29.944,155.618
C05180=1055.495,-10.480,429.330,171.022,29.946,155.618
C05181=1055.501,-10.230,429.317,171.024,29.948,155.619
C05182=1055.508,-9.981,429.302,171.025,29.950,155.619
C05183=1055.513,-9.731,429.288,171.026,29.952,155.619
C05184=1055.520,-9.482,429.274,171.028,29.954,155.619
C05185=1055.526,-9.232,429.260,171.030,29.956,155.620
C05186=1055.532,-8.983,429.245,171.032,29.958,155.620
C05187=1055.539,-8.733,429.231,171.034,29.960,155.620
C05188=1055.545,-8.484,429.217,171.035,29.963,155.620
C05189=1055.551,-8.233,429.203,171.037,29.965,155.621
C05190=1055.557,-7.985,429.188,171.038,29.967,155.621
C05191=1055.564,-7.735,429.174,171.040,29.968,155.621
C05192=1055.569,-7.486,429.160,171.041,29.970,155.622
C05193=1055.576,-7.236,429.145,171.043,29.973,155.622
C05194=1055.582,-6.987,429.132,171.045,29.975,155.622
C05195=1055.588,-6.737,429.117,171.047,29.977,155.622
C05196=1055.595,-6.487,429.102,171.049,29.979,155.623
C05197=1055.600,-6.238,429.088,171.049,29.981,155.623
C05198=1055.607,-5.988,429.074,171.051,29.983,155.623
C05199=1055.613,-5.739,429.060,171.053,29.985,155.623
C05200=1055.619,-5.489,429.045,171.055,29.987,155.624
C05201=1055.626,-5.241,429.031,171.056,29.989,155.624
C05202=1055.632,-4.990,429.017,171.058,29.991,155.624
C05203=1055.638,-4.741,429.002,171.060,29.994,155.624
C05204=1055.644,-4.492,428.987,171.061,29.996,155.625
C05205=1055.651,-4.242,428.973,171.063,29.998,155.625
C05206=1055.657,-3.992,428.958,171.064,30.000,155.625
C05207=1055.663,-3.743,428.944,171.066,30.001,155.625
C05208=1055.669,-3.493,428.930,171.068,30.004,155.626
C05209=1055.675,-3.244,428.916,171.070,30.006,155.626
C05210=1055.681,-2.994,428.900,171.072,30.008,155.626
C05211=1055.688,-2.712,428.884,171.073,30.011,155.627
C05212=1055.695,-2.430,428.867,171.075,30.013,155.627
C05213=1055.702,-2.148,428.851,171.077,30.016,155.627
C05214=1055.709,-1.866,428.834,171.079,30.018,155.628
C05215=1055.714,-1.616,428.820,171.080,30.020,155.628
C05216=1055.721,-1.367,428.805,171.081,30.022,155.628
C05217=1055.726,-1.118,428.790,171.083,30.024,155.628
C05218=1055.733,-0.868,428.776,171.085,30.026,155.629
C05219=1055.739,-0.618,428.761,171.086,30.028,155.629
C05220=1055.745,-0.369,428.747,171.088,30.031,155.629
C05221=1055.751,-0.119,428.732,171.090,30.033,155.630
C05222=1055.758,0.130,428.717,171.091,30.035,155.630
C05223=1055.763,0.379,428.702,171.093,30.038,155.630
C05224=1055.770,0.629,428.687,171.094,30.040,155.631
C05225=1055.775,0.878,428.673,171.096,30.042,155.631
C05226=1055.782,1.128,428.658,171.098,30.044,155.631
C05227=1055.788,1.378,428.644,171.100,30.046,155.631
C05228=1055.794,1.627,428.629,171.100,30.048,155.632
C05229=1055.800,1.877,428.614,171.102,30.050,155.632
C05230=1055.806,2.126,428.599,171.104,30.053,155.632
C05231=1055.812,2.375,428.584,171.106,30.055,155.633
C05232=1055.818,2.625,428.569,171.108,30.057,155.633
C05233=1055.824,2.875,428.554,171.109,30.059,155.633
C05234=1055.830,3.124,428.539,171.110,30.061,155.633
C05235=1055.836,3.373,428.524,171.112,30.064,155.634
C05236=1055.843,3.623,428.510,171.114,30.066,155.634
C05237=1055.849,3.872,428.495,171.115,30.068,155.634
C05238=1055.855,4.122,428.480,171.117,30.070,155.635
C05239=1055.861,4.371,428.465,171.118,30.072,155.635
C05240=1055.867,4.620,428.450,171.120,30.074,155.635
C05241=1055.874,4.870,428.436,171.122,30.077,155.635
C05242=1055.880,5.120,428.421,171.123,30.079,155.636
C05243=1055.886,5.369,428.406,171.125,30.081,155.636
C05244=1055.892,5.618,428.391,171.127,30.083,155.636
C05245=1055.898,5.868,428.376,171.128,30.085,155.637
C05246=1055.905,6.117,428.361,171.130,30.087,155.637
C05247=1055.910,6.367,428.346,171.131,30.089,155.637
C05248=1055.916,6.616,428.331,171.133,30.092,155.638
C05249=1055.923,6.866,428.316,171.135,30.094,155.638
C05250=1055.929,7.116,428.301,171.136,30.096,155.638
C05251=1055.935,7.365,428.286,171.137,30.098,155.638
C05252=1055.941,7.614,428.272,171.139,30.101,155.639
C05253=1055.948,7.864,428.257,171.141,30.103,155.639
C05254=1055.954,8.114,428.242,171.143,30.105,155.639
C05255=1055.960,8.363,428.227,171.144,30.107,155.640
C05256=1055.966,8.612,428.212,171.145,30.109,155.640
C05257=1055.972,8.862,428.197,171.147,30.111,155.640
C05258=1055.978,9.112,428.182,171.149,30.113,155.640
C05259=1055.985,9.361,428.166,171.151,30.115,155.641
C05260=1055.991,9.611,428.151,171.152,30.118,155.641
C05261=1055.997,9.860,428.137,171.153,30.120,155.641
C05262=1056.003,10.109,428.122,171.155,30.122,155.642
C05263=1056.010,10.359,428.107,171.157,30.124,155.642
C05264=1056.016,10.609,428.092,171.159,30.127,155.642
C05265=1056.022,10.858,428.076,171.160,30.129,155.643
C05266=1056.028,11.107,428.061,171.161,30.131,155.643
C05267=1056.034,11.356,428.046,171.163,30.133,155.643
C05268=1056.041,11.606,428.031,171.165,30.135,155.643
C05269=1056.047,11.856,428.016,171.167,30.137,155.644
C05270=1056.053,12.105,428.001,171.168,30.139,155.644
C05271=1056.060,12.354,427.985,171.169,30.141,155.644
C05272=1056.066,12.604,427.970,171.171,30.144,155.645
C05273=1056.072,12.853,427.955,171.173,30.146,155.645
C05274=1056.078,13.103,427.940,171.175,30.148,155.645
C05275=1056.086,13.387,427.923,171.176,30.151,155.645
C05276=1056.093,13.671,427.906,171.178,30.153,155.646
C05277=1056.100,13.956,427.888,171.180,30.156,155.646
C05278=1056.106,14.239,427.871,171.182,30.158,155.647
C05279=1056.113,14.488,427.856,171.183,30.160,155.647
C05280=1056.119,14.738,427.841,171.185,30.163,155.647
C05281=1056.125,14.987,427.824,171.186,30.165,155.647
C05282=1056.132,15.237,427.810,171.188,30.167,155.648
C05283=1056.138,15.487,427.795,171.189,30.169,155.648
C05284=1056.143,15.735,427.779,171.191,30.172,155.648
C05285=1056.150,15.985,427.764,171.192,30.174,155.649
C05286=1056.156,16.235,427.749,171.194,30.176,155.649
C05287=1056.162,16.484,427.733,171.196,30.178,155.649
C05288=1056.168,16.734,427.718,171.197,30.181,155.650
C05289=1056.174,16.984,427.702,171.199,30.183,155.650
C05290=1056.181,17.233,427.686,171.200,30.185,155.650
C05291=1056.187,17.482,427.671,171.202,30.188,155.651
C05292=1056.192,17.731,427.656,171.204,30.190,155.651
C05293=1056.199,17.981,427.641,171.205,30.192,155.651
C05294=1056.205,18.230,427.624,171.206,30.194,155.651
C05295=1056.211,18.480,427.609,171.208,30.197,155.652
C05296=1056.218,18.729,427.594,171.210,30.199,155.652
C05297=1056.223,18.979,427.578,171.211,30.201,155.652
C05298=1056.230,19.228,427.563,171.213,30.203,155.653
C05299=1056.236,19.478,427.547,171.214,30.205,155.653
C05300=1056.242,19.727,427.532,171.216,30.208,155.653
C05301=1056.249,19.976,427.516,171.218,30.210,155.654
C05302=1056.255,20.226,427.501,171.219,30.212,155.654
C05303=1056.261,20.475,427.486,171.220,30.214,155.654
C05304=1056.266,20.725,427.470,171.222,30.217,155.655
C05305=1056.273,20.974,427.454,171.224,30.219,155.655
C05306=1056.279,21.224,427.439,171.226,30.221,155.655
C05307=1056.285,21.473,427.423,171.227,30.224,155.656
C05308=1056.291,21.723,427.408,171.228,30.226,155.656
C05309=1056.298,21.972,427.392,171.230,30.228,155.656
C05310=1056.303,22.222,427.376,171.232,30.231,155.657
C05311=1056.309,22.471,427.360,171.233,30.233,155.657
C05312=1056.316,22.720,427.344,171.234,30.235,155.657
C05313=1056.322,22.970,427.329,171.236,30.237,155.657
C05314=1056.328,23.219,427.313,171.238,30.240,155.658
C05315=1056.334,23.469,427.298,171.240,30.242,155.658
C05316=1056.341,23.718,427.282,171.240,30.244,155.658
C05317=1056.346,23.968,427.267,171.242,30.247,155.659
C05318=1056.353,24.217,427.251,171.244,30.249,155.659
C05319=1056.359,24.466,427.235,171.246,30.251,155.659
C05320=1056.365,24.716,427.220,171.248,30.253,155.660
C05321=1056.371,24.965,427.203,171.248,30.256,155.660
C05322=1056.377,25.215,427.187,171.250,30.258,155.660
C05323=1056.384,25.464,427.172,171.252,30.260,155.661
C05324=1056.389,25.714,427.156,171.254,30.263,155.661
C05325=1056.396,25.963,427.140,171.255,30.265,155.661
C05326=1056.402,26.213,427.125,171.256,30.267,155.662
C05327=1056.409,26.462,427.109,171.258,30.269,155.662
C05328=1056.414,26.711,427.093,171.260,30.272,155.662
C05329=1056.420,26.961,427.077,171.261,30.274,155.663
C05330=1056.427,27.210,427.062,171.262,30.276,155.663
C05331=1056.433,27.460,427.045,171.264,30.278,155.663
C05332=1056.439,27.709,427.030,171.266,30.281,155.664
C05333=1056.445,27.959,427.014,171.267,30.283,155.664
C05334=1056.451,28.208,426.998,171.269,30.285,155.664
C05335=1056.458,28.457,426.982,171.270,30.287,155.665
C05336=1056.464,28.706,426.966,171.272,30.290,155.665
C05337=1056.469,28.956,426.950,171.273,30.292,155.665
C05338=1056.475,29.206,426.934,171.275,30.294,155.666
C05339=1056.483,29.491,426.917,171.276,30.297,155.666
C05340=1056.490,29.776,426.898,171.278,30.300,155.666
C05341=1056.497,30.061,426.879,171.280,30.302,155.667
C05342=1056.504,30.347,426.861,171.282,30.305,155.667
C05343=1056.509,30.596,426.845,171.284,30.307,155.667
C05344=1056.516,30.845,426.829,171.285,30.309,155.668
C05345=1056.522,31.095,426.814,171.286,30.312,155.668
C05346=1056.528,31.345,426.797,171.288,30.314,155.668
C05347=1056.534,31.594,426.781,171.290,30.317,155.669
C05348=1056.540,31.843,426.765,171.291,30.319,155.669
C05349=1056.546,32.092,426.749,171.292,30.321,155.669
C05350=1056.552,32.342,426.733,171.294,30.324,155.670
C05351=1056.558,32.591,426.717,171.296,30.326,155.670
C05352=1056.564,32.841,426.701,171.298,30.329,155.671
C05353=1056.571,33.091,426.685,171.298,30.331,155.671
C05354=1056.577,33.340,426.669,171.300,30.333,155.671
C05355=1056.583,33.589,426.653,171.302,30.336,155.672
C05356=1056.589,33.839,426.636,171.304,30.338,155.672
C05357=1056.595,34.088,426.620,171.305,30.340,155.672
C05358=1056.602,34.337,426.604,171.306,30.342,155.673
C05359=1056.608,34.586,426.588,171.308,30.344,155.673
C05360=1056.614,34.836,426.572,171.310,30.347,155.673
C05361=1056.620,35.085,426.556,171.311,30.349,155.674
C05362=1056.626,35.335,426.539,171.313,30.351,155.674
C05363=1056.632,35.585,426.523,171.314,30.354,155.674
C05364=1056.639,35.834,426.507,171.316,30.356,155.674
C05365=1056.645,36.083,426.491,171.317,30.358,155.675
C05366=1056.651,36.332,426.475,171.319,30.361,155.675
C05367=1056.657,36.582,426.458,171.321,30.363,155.675
C05368=1056.663,36.831,426.442,171.322,30.366,155.676
C05369=1056.670,37.081,426.426,171.323,30.368,155.676
C05370=1056.676,37.330,426.410,171.325,30.370,155.676
C05371=1056.682,37.579,426.393,171.327,30.373,155.677
C05372=1056.688,37.829,426.377,171.328,30.375,155.677
C05373=1056.694,38.078,426.361,171.329,30.377,155.678
C05374=1056.700,38.327,426.345,171.331,30.379,155.678
C05375=1056.706,38.577,426.328,171.333,30.382,155.678
C05376=1056.712,38.827,426.312,171.335,30.384,155.679
C05377=1056.718,39.076,426.295,171.335,30.387,155.679
C05378=1056.724,39.325,426.279,171.337,30.389,155.679
C05379=1056.730,39.574,426.262,171.339,30.392,155.680
C05380=1056.736,39.824,426.246,171.340,30.394,155.680
C05381=1056.742,40.073,426.230,171.342,30.396,155.680
C05382=1056.749,40.323,426.213,171.343,30.399,155.681
C05383=1056.755,40.572,426.197,171.345,30.401,155.681
C05384=1056.761,40.821,426.180,171.346,30.403,155.681
C05385=1056.767,41.070,426.164,171.348,30.405,155.682
C05386=1056.773,41.320,426.147,171.350,30.408,155.682
C05387=1056.779,41.569,426.131,171.351,30.410,155.682
C05388=1056.785,41.819,426.115,171.352,30.413,155.683
C05389=1056.790,42.069,426.098,171.354,30.415,155.683
C05390=1056.797,42.318,426.081,171.356,30.418,155.683
C05391=1056.803,42.567,426.064,171.357,30.420,155.684
C05392=1056.809,42.817,426.048,171.358,30.422,155.684
C05393=1056.815,43.066,426.032,171.360,30.424,155.684
C05394=1056.821,43.315,426.015,171.362,30.427,155.685
C05395=1056.827,43.564,425.998,171.363,30.429,155.685
C05396=1056.833,43.814,425.982,171.364,30.432,155.686
C05397=1056.840,44.064,425.965,171.366,30.434,155.686
C05398=1056.845,44.313,425.948,171.368,30.437,155.686
C05399=1056.851,44.562,425.932,171.369,30.439,155.687
C05400=1056.857,44.812,425.915,171.371,30.441,155.687
C05401=1056.864,45.060,425.898,171.372,30.444,155.687
C05402=1056.869,45.311,425.881,171.373,30.446,155.688
C05403=1056.877,45.596,425.862,171.375,30.449,155.688
C05404=1056.883,45.881,425.843,171.377,30.452,155.688
C05405=1056.890,46.166,425.824,171.378,30.455,155.689
C05406=1056.897,46.451,425.805,171.380,30.458,155.689
C05407=1056.902,46.701,425.789,171.382,30.460,155.690
C05408=1056.909,46.950,425.771,171.384,30.462,155.690
C05409=1056.915,47.200,425.755,171.385,30.464,155.690
C05410=1056.920,47.449,425.737,171.386,30.467,155.691
C05411=1056.926,47.698,425.721,171.388,30.470,155.691
C05412=1056.933,47.948,425.704,171.390,30.472,155.691
C05413=1056.939,48.197,425.688,171.391,30.475,155.692
C05414=1056.944,48.446,425.671,171.393,30.477,155.692
C05415=1056.951,48.695,425.654,171.394,30.479,155.693
C05416=1056.957,48.945,425.637,171.396,30.482,155.693
C05417=1056.963,49.194,425.620,171.397,30.484,155.693
C05418=1056.969,49.444,425.603,171.399,30.487,155.694
C05419=1056.975,49.693,425.587,171.401,30.489,155.694
C05420=1056.981,49.943,425.569,171.401,30.492,155.694
C05421=1056.987,50.192,425.553,171.403,30.494,155.695
C05422=1056.993,50.441,425.536,171.405,30.496,155.695
C05423=1056.999,50.691,425.519,171.407,30.499,155.695
C05424=1057.005,50.940,425.502,171.408,30.501,155.696
C05425=1057.011,51.189,425.485,171.409,30.504,155.696
C05426=1057.017,51.439,425.467,171.411,30.506,155.696
C05427=1057.023,51.688,425.451,171.412,30.508,155.697
C05428=1057.029,51.937,425.434,171.414,30.511,155.697
C05429=1057.036,52.186,425.417,171.415,30.513,155.698
C05430=1057.041,52.436,425.400,171.417,30.515,155.698
C05431=1057.048,52.685,425.383,171.418,30.518,155.698
C05432=1057.053,52.935,425.366,171.420,30.521,155.699
C05433=1057.060,53.184,425.349,171.422,30.523,155.699
C05434=1057.066,53.433,425.333,171.422,30.525,155.699
C05435=1057.072,53.683,425.315,171.424,30.527,155.700
C05436=1057.078,53.932,425.298,171.426,30.530,155.700
C05437=1057.084,54.181,425.281,171.428,30.532,155.700
C05438=1057.090,54.431,425.264,171.429,30.535,155.701
C05439=1057.096,54.680,425.247,171.430,30.537,155.701
C05440=1057.102,54.929,425.230,171.432,30.540,155.701
C05441=1057.108,55.179,425.212,171.434,30.542,155.702
C05442=1057.114,55.428,425.196,171.435,30.544,155.702
C05443=1057.121,55.677,425.179,171.437,30.547,155.703
C05444=1057.126,55.927,425.162,171.438,30.549,155.703
C05445=1057.133,56.176,425.145,171.439,30.552,155.703
C05446=1057.139,56.426,425.127,171.441,30.554,155.704
C05447=1057.145,56.675,425.111,171.443,30.557,155.704
C05448=1057.152,56.924,425.093,171.445,30.559,155.704
C05449=1057.157,57.173,425.076,171.445,30.561,155.705
C05450=1057.163,57.422,425.059,171.447,30.563,155.705
C05451=1057.170,57.672,425.042,171.449,30.566,155.705
C05452=1057.175,57.921,425.025,171.451,30.568,155.706
C05453=1057.182,58.171,425.007,171.452,30.571,155.706
C05454=1057.187,58.420,424.991,171.453,30.573,155.706
C05455=1057.194,58.670,424.973,171.455,30.576,155.707
C05456=1057.201,58.918,424.956,171.456,30.578,155.707
C05457=1057.207,59.168,424.938,171.458,30.580,155.708
C05458=1057.213,59.418,424.922,171.460,30.583,155.708
C05459=1057.219,59.667,424.904,171.461,30.585,155.708
C05460=1057.225,59.916,424.887,171.462,30.588,155.709
